(* IEC 61131-3 sources: elnaProjects/ElpcLogic/PomarKc7Changed/build_USO_ecl/_, 1 file *)

(* ---- plc.st ---- *)
TYPE
  TYPE_DualStateImAction : (_on, _off);
  TYPE_PhaseAlgoritmAction : (_run, _reset);
  TYPE_basketStats : STRUCT
    BASKET_NOTDEFINED : BYTE := 0;
    BASKET_ROLLEDIN : BYTE := 1;
    BASKET_ROLLEDOUT : BYTE := 2;
    BASKET_TRANSITIONAL : BYTE := 3;
    BASKET_ERROR : BYTE := 4;
    BASKET_TEST : BYTE := 5;
  END_STRUCT;
  TYPE_Answers : STRUCT
    ANS_NONE : UINT := 0;
    ANS_YES : UINT := 1;
    ANS_NO : UINT := 2;
    ANS_CANCEL : UINT := 4;
    ANS_RETRY : UINT := 8;
  END_STRUCT;
  struct_OilPump : STRUCT
    inCommand : WORD;
    inCommand_Alg : WORD;
    inCommand_ARM : WORD;
    status : DWORD;
    onStatus : BYTE;
    inOpcCommandsDisabled : BOOL;
    sdvig : BOOL;
    Ns : BOOL;
    CommandFault : BOOL;
    Accident : BOOL;
    Local : BOOL;
    Distance : BOOL;
    BreakCmdOn : BOOL;
    BreakCmdOff : BOOL;
    OpcCommandsDisabled : BOOL;
    lastCmdIsOn : BOOL;
    ISVALIDREF_statOn : BOOL;
    ISVALIDREF_statOff : BOOL;
    ISVALIDREF_cmdOn : BOOL;
    ISVALIDREF_cmdOff : BOOL;
    ISVALIDREF_inBreakCmdOn : BOOL;
    ISVALIDREF_inBreakCmdOff : BOOL;
    inBlocked : BOOL;
    Blocked : BOOL;
    Osnovnoy : BOOL;
    Rezervny : BOOL;
    cmdOn : BOOL;
    cmdOff : BOOL;
    reliability : BOOL;
  END_STRUCT;
  struct_AlgTimers : STRUCT
    AutoPns_OffTimer : UINT;
    AutoPns_OnTimer : UINT;
    vibegPNS_Timer : UINT;
    NO_waitCloseKran : UINT;
    AO_waitKran : UINT;
    testPms_BreakTest : UINT;
    testdPmg_BreakTest : UINT;
    puskOilSystem_BreakPuskTimer_Poil : UINT;
    engineRun_BreakPuskTimer : UINT;
    filling_BreakPuskTimer : UINT;
    filling_waitAfterKran4 : UINT;
    filling_waitAfterKran5 : UINT;
    puskK_wait720 : UINT;
    puskV_wait600 : UINT;
    No_wait120 : UINT;
    No_wait600 : UINT;
    No_wait5 : UINT;
  END_STRUCT;
  struct_Question : STRUCT
    AnswerVariants : UINT;
    inCommand : WORD;
    ask : BOOL;
    reset : BOOL;
    status : DWORD;
    answer : UINT;
    OpcCommandsDisabled : BOOL;
    inOpcCommandsDisabled : BOOL;
  END_STRUCT;
  AlgoritmsQuestions : STRUCT
    vibegPNS_algContinue : struct_Question;
    testPms_algContinue : struct_Question;
    testdPmg_algContinue : struct_Question;
    puskK_questionFilling : struct_Question;
    puskK_questionUnload : struct_Question;
    puskV_questionEngine : struct_Question;
    puskV_questionMVoff : struct_Question;
    SemiAutoPusk_cmdRun1ph : struct_Question;
    SemiAutoPusk_cmdRun2ph : struct_Question;
    SemiAutoPusk_cmdRun3ph : struct_Question;
    SemiAutoPusk_cmdRun4ph : struct_Question;
  END_STRUCT;
  TYPE_commandDualInput : STRUCT
    CMD_ON : BYTE := 1;
    CMD_OFF : BYTE := 2;
    CMD_RESET : BYTE := 3;
  END_STRUCT;
  TYPE_CommandAnalog : STRUCT
    cmd_SetUstavki : WORD := 1;
    cmd_SetRemont : WORD := 2;
    cmd_ResetRemont : WORD := 3;
    cmd_kvitNotReliable : WORD := 4;
  END_STRUCT;
  struct_AnalogParametr : STRUCT
    inCommand : WORD;
    inCommand_Alg : WORD;
    inCommand_ARM : WORD;
    status : DWORD;
    newValue : LREAL;
    currentValue : LREAL;
    minVal : LREAL;
    maxVal : LREAL;
    maxStep : LREAL;
    minVal_ISVALIDREF : BOOL;
    maxVal_ISVALIDREF : BOOL;
    maxStep_ISVALIDREF : BOOL;
    inOpcCommandsDisabled : BOOL;
    Value : LREAL;
    isValidValue : BOOL;
    OpcCommandsDisabled : BOOL;
  END_STRUCT;
  struct_AI : STRUCT
    value : LREAL;
    status : DWORD;
    interval : BYTE;
    inCommand : WORD;
    blConnect : BOOL;
    dLL : LREAL;
    dHL : LREAL;
    dLA : LREAL;
    dHA : LREAL;
    dLW : LREAL;
    dHW : LREAL;
    LL : LREAL;
    HL : LREAL;
    LA : LREAL;
    HA : LREAL;
    LW : LREAL;
    HW : LREAL;
    ISVALIDREF_LA : BOOL;
    ISVALIDREF_HA : BOOL;
    ISVALIDREF_LW : BOOL;
    ISVALIDREF_HW : BOOL;
    inpLL : LREAL;
    inpHL : LREAL;
    CurrentShotCircuit : LREAL;
    CurrentBreakCircuit : LREAL;
    maxChangeSpeed : LREAL;
    maxChangeSpeedDown : LREAL;
    ChangeSpeed : LREAL;
    histeresis : LREAL;
    aperturFilter : LREAL;
    exponentialFilter : LREAL;
    rassoglasovanie : LREAL;
    OpcCommandsDisabled : BOOL;
    Disabled_LA : BOOL;
    Disabled_HA : BOOL;
    Disabled_LW : BOOL;
    Disabled_HW : BOOL;
    delayLA : TIME;
    delayLW : TIME;
    delayHW : TIME;
    delayHA : TIME;
    minValue_ISVALIDREF : BOOL;
    maxValue_ISVALIDREF : BOOL;
    minValue : LREAL;
    maxValue : LREAL;
    inOpcCommandsDisabled : BOOL;
    imit : BOOL;
    remont : BOOL;
    NS : BOOL;
    NS_Min : BOOL;
    NS_Max : BOOL;
    inCommand_Alg : WORD;
    inCommand_ARM : WORD;
    dMaxChangeSpeed : LREAL;
    dMaxChangeSpeedDown : LREAL;
  END_STRUCT;
  AiConfig : STRUCT
    Tstali_statora_kanal_1 : struct_AI;
    Tstali_statora_kanal_2 : struct_AI;
    Tstali_statora_kanal_3 : struct_AI;
    Tmedi_statora_kanal_1 : struct_AI;
    Tmedi_statora_kanal_2 : struct_AI;
    Tmedi_statora_kanal_3 : struct_AI;
    Toporno_podshipnika_EDT_1 : struct_AI;
    Toy_podshipnika_EDT_2 : struct_AI;
    Toy_podshipnika_kol_EDT_3 : struct_AI;
    Toy_podshipnika_kol_EDT_4 : struct_AI;
    Toy_podshipnika_shest_red_EDT_5 : struct_AI;
    Ty_podshipnika_red_EDT_6 : struct_AI;
    Ty_podshipnika_nagnet_EDT_7_1 : struct_AI;
    Ty_podshipnika_nagnet_EDT_7_2 : struct_AI;
    Toy_podshipnika_svobod_konca_EDT_8_1 : struct_AI;
    Toy_podshipnika_svobod_konca_EDT_8_2 : struct_AI;
    Toy_podshipnika_rab_kol_EDT_9_1 : struct_AI;
    Toy_podshipnika_rab_kol_EDT_9_2 : struct_AI;
    Toy_podshipnika_nerab_kol_EDT_10_1 : struct_AI;
    Toy_podshipnika_nerab_kol_EDT_10_2 : struct_AI;
    Tholodnogo_vozduha_ED_kanal_1 : struct_AI;
    Tholodnogo_vozduha_ED_kanal_2 : struct_AI;
    Tgorjachego_vozduha_ED_kanal_1 : struct_AI;
    Tgorjachego_vozduha_ED_kanal_2 : struct_AI;
    Tnarujnogo_vozduha : struct_AI;
    Tgaza_na_vhode_H : struct_AI;
    Tgaza_na_vyhode_H : struct_AI;
    Tmasla_do_AVOM : struct_AI;
    Tmasla_posle_AVOM : struct_AI;
    Tmasla_MB : struct_AI;
    Tmasla_MB_TEN : struct_AI;
    Tshu : struct_AI;
    Pmaslo_sm_nizkoe : struct_AI;
    Pmaslo_sm_vysokoe : struct_AI;
    Pmasla_posle_GNS : struct_AI;
    Pmasla_posle_NU : struct_AI;
    Pgaza_na_vhode_nagnetatelia : struct_AI;
    Pgaza_na_vyhode_nagnetatelia : struct_AI;
    Pimpuls_gaz : struct_AI;
    dPgaza_na_maslo_filtre : struct_AI;
    dPgaza_na_konfuzore : struct_AI;
    dPmaslo_gaz : struct_AI;
    Os_sdvig_nagnetatelja_plus : struct_AI;
    Os_sdvig_nagnetatelja_minus : struct_AI;
    Yroven_masla_MB : struct_AI;
    Kontrol_per_220V : struct_AI;
    Kontrol_post_220V : struct_AI;
    Tok_statora : struct_AI;
    Vibro_skorost_OPED_T1 : struct_AI;
    Vibro_skorost_OYPED_T2 : struct_AI;
    Vibro_skorost_OYP_kolesa_ED_T3 : struct_AI;
    Vibro_skorost_OP_kolesa_RH_T4 : struct_AI;
    Vibro_skorost_OP_shesterni_RED_T5 : struct_AI;
    Vibro_skorost_OP_shesterni_RED_T6 : struct_AI;
  END_STRUCT;
  struct_singleOutput : STRUCT
    wait_time : TIME;
    inCommand : WORD;
    inOpcCommandsDisabled : BOOL;
    Q : BOOL;
    status : DWORD;
    OpcCommandsDisabled : BOOL;
    inCommand_Alg : WORD;
    inCommand_ARM : WORD;
  END_STRUCT;
  IM_singleOutputs : STRUCT
    Rabota_EGPA : struct_singleOutput;
    Neispr_EGPA : struct_singleOutput;
    Avary_EGPA : struct_singleOutput;
    U_lamp_SHU : struct_singleOutput;
    AO_knopka_ind : struct_singleOutput;
    Pusk_SHUP : struct_singleOutput;
    Stop_SHUP : struct_singleOutput;
    NO_fonar : struct_singleOutput;
    PC_fonar : struct_singleOutput;
    AC_fonar : struct_singleOutput;
    Kr1_smazka : struct_singleOutput;
    Kr2_smazka : struct_singleOutput;
    Kr4_open_from_alg : struct_singleOutput;
    Synch_rej_K1 : struct_singleOutput;
  END_STRUCT;
  struct_Alg : STRUCT
    inRunOnStart : BOOL;
    inCanRun : BOOL;
    inHasError : BOOL;
    inEnded : BOOL;
    inOpcCommandsDisabled : BOOL;
    inCommand : WORD;
    inCommand_ARM : WORD;
    inCommand_Alg : WORD;
    status : DWORD;
    CanRun : BOOL;
    OpcCommandsDisabled : BOOL;
    isRuning : BOOL;
    HasError : BOOL;
    isEnded : BOOL;
    RunOnStart : BOOL;
    Start : DWORD;
    Error : DWORD;
    Top : DWORD;
  END_STRUCT;
  AlgoritmsConfig : STRUCT
    autoNu : struct_Alg;
    AutoPns : struct_Alg;
    AutoAvom : struct_Alg;
    AutoTen : struct_Alg;
    AntiPompag : struct_Alg;
    testIm : struct_Alg;
    TestProtection : struct_Alg;
    Remont : struct_Alg;
    ppu : struct_Alg;
    puskOilSystem : struct_Alg;
    engineRun : struct_Alg;
    filling : struct_Alg;
    LineToRing : struct_Alg;
    RingToLine : struct_Alg;
    Apusk : struct_Alg;
    SemiAutoPusk : struct_Alg;
    no : struct_Alg;
    vibegPNS : struct_Alg;
    ao : struct_Alg;
    testPms : struct_Alg;
    testdPmg : struct_Alg;
    puskV : struct_Alg;
    puskK : struct_Alg;
    Pusk_F_faza1 : struct_Alg;
    Pusk_F_faza2 : struct_Alg;
    Pusk_TH_faza : struct_Alg;
    Prov_PMS_ALG : struct_Alg;
    Prov_opressovka_ALG : struct_Alg;
    Pusk_SEC_faza_chastotny : struct_Alg;
    Pusk_SEC_faza_reactor : struct_Alg;
  END_STRUCT;
  TItemDIN : STRUCT
    wFlags : UINT := 0;
    wValue : UINT := 0;
    nanosec : ULINT := 0;
    reserve : ULINT := 0;
  END_STRUCT;
  TItemAIN : STRUCT
    wFlags : UINT := 0;
    wReserved : UINT := 0;
    dblValue : LREAL := 0.0;
    nanosec : ULINT := 0;
    reserve : ULINT := 0;
  END_STRUCT;
  struct_ReserveIM : STRUCT
    var1 : BOOL;
    var2 : BOOL;
  END_STRUCT;
  TYPE_ReliableBit : STRUCT
    value : BOOL;
    reliability : BOOL;
    _inversed : BOOL;
  END_STRUCT;
  struct_DI : STRUCT
    imit : BOOL;
    value : WORD;
    reliability : WORD;
    bits : ARRAY [0..15] OF TYPE_ReliableBit;
    blConnect : BOOL;
  END_STRUCT;
  struct_Kran : STRUCT
    inCommand : WORD;
    status : DWORD;
    onStatus : BYTE;
    inOpcCommandsDisabled : BOOL;
    sdvig : BOOL;
    Ns : BOOL;
    Dp : BOOL;
    CommandFault : BOOL;
    Accident : BOOL;
    Auto : BOOL;
    Manual : BOOL;
    Local : BOOL;
    Distance : BOOL;
    ErrorPowerOff : BOOL;
    ErrorBlock : BOOL;
    So : BOOL;
    Sz : BOOL;
    OpcCommandsDisabled : BOOL;
    lastCmdIsOn : BOOL;
    ISVALIDREF_statOn : BOOL;
    ISVALIDREF_statOff : BOOL;
    ISVALIDREF_cmdOn : BOOL;
    ISVALIDREF_cmdOff : BOOL;
    ISVALIDREF_inSo : BOOL;
    ISVALIDREF_inSz : BOOL;
    ISVALIDREF_inDp : BOOL;
    continueHoldCommand : TIME;
    inCommand_Alg : WORD;
    inCommand_ARM : WORD;
    cmdOn : BOOL;
    cmdOff : BOOL;
    reliability : BOOL;
  END_STRUCT;
  struct_Switch : STRUCT
    inCommand : WORD;
    status : DWORD;
    onStatus : BYTE;
    inOpcCommandsDisabled : BOOL;
    sdvig : BOOL;
    Ns : BOOL;
    CommandFault : BOOL;
    Accident : BOOL;
    Auto : BOOL;
    Manual : BOOL;
    Local : BOOL;
    Distance : BOOL;
    ErrorPowerOff : BOOL;
    ErrorBlock : BOOL;
    BreakCmdOn : BOOL;
    BreakCmdOff : BOOL;
    OpcCommandsDisabled : BOOL;
    lastCmdIsOn : BOOL;
    ISVALIDREF_statOn : BOOL;
    ISVALIDREF_statOff : BOOL;
    ISVALIDREF_cmdOn : BOOL;
    ISVALIDREF_cmdOff : BOOL;
    ISVALIDREF_inBreakCmdOn : BOOL;
    ISVALIDREF_inBreakCmdOff : BOOL;
    inCommand_Alg : WORD;
    inCommand_ARM : WORD;
    cmdOn : BOOL;
    cmdOff : BOOL;
    reliability : BOOL;
  END_STRUCT;
  struct_SectionSwitch : STRUCT
    inCommand : WORD;
    status : DWORD;
    onStatus : BYTE;
    inOpcCommandsDisabled : BOOL;
    sdvig : BOOL;
    Ns : BOOL;
    CommandFault : BOOL;
    Accident : BOOL;
    Local : BOOL;
    Distance : BOOL;
    OpcCommandsDisabled : BOOL;
    lastCmdIsOn : BOOL;
    offKNA : BOOL;
    basketStatus : BYTE;
    ISVALIDREF_statOn : BOOL;
    ISVALIDREF_statOff : BOOL;
    ISVALIDREF_cmdOn : BOOL;
    ISVALIDREF_cmdOff : BOOL;
    ISVALIDREF_inBreakCmdOn : BOOL;
    ISVALIDREF_inBreakCmdOff : BOOL;
    BreakCmdOn : BOOL;
    BreakCmdOff : BOOL;
    ISVALIDREF_basketRolledIn : BOOL;
    ISVALIDREF_basketRolledOut : BOOL;
    ISVALIDREF_basketTest : BOOL;
    inCommand_Alg : WORD;
    inCommand_ARM : WORD;
    cmdOn : BOOL;
    cmdOff : BOOL;
    reliability : BOOL;
  END_STRUCT;
  struct_ReserveIM2 : STRUCT
    var1 : BOOL;
    var2 : BOOL;
  END_STRUCT;
  struct_singleSignal : STRUCT
    reliability : BOOL;
    inverse : BOOL;
    DelayOn : TIME;
    DelayOff : TIME;
    Q : BOOL;
    status : DWORD;
    Disabled_Sig : BOOL;
  END_STRUCT;
  IM_singleSignals : STRUCT
    dP_maslo_gaz_Less100 : struct_singleSignal;
    dp_kran1_Less100 : struct_singleSignal;
    Razreshenie_zagruzki_dvig : struct_singleSignal;
    Vozbud_gotovnost : struct_singleSignal;
    Vozbud_neispr_tsepey_upr_AVR_pit : struct_singleSignal;
    Vozbud_neispravnost : struct_singleSignal;
    SHAVR1_v_rabote : struct_singleSignal;
    SHAVR2_v_rabote : struct_singleSignal;
    Avariinoe_otkluch_vikluchatelya : struct_singleSignal;
    Assinhronnii_hod_peregruzka : struct_singleSignal;
    SHU_v_GPA_vkluch : struct_singleSignal;
    SHP_v_GPA_vkluch : struct_singleSignal;
    QF1_on : struct_singleSignal;
    QF2_on : struct_singleSignal;
    QF23_on : struct_singleSignal;
    QF4_QF5_on : struct_singleSignal;
    QF6_QF7_on : struct_singleSignal;
    QF8_QF9_on : struct_singleSignal;
    QF10_QF11_on : struct_singleSignal;
    QF12_QF13_on : struct_singleSignal;
    QF14_QF15_on : struct_singleSignal;
    QF22_on : struct_singleSignal;
    NS_G1_G2 : struct_singleSignal;
    NS_G3_G4 : struct_singleSignal;
    NS_G15_G16 : struct_singleSignal;
    NS_G17 : struct_singleSignal;
    NS_G5_G6 : struct_singleSignal;
    NS_G7_G8 : struct_singleSignal;
    NS_G18_G19 : struct_singleSignal;
    NS_G10_G11 : struct_singleSignal;
    NS_G13_G14 : struct_singleSignal;
    Uroven_masla_akkum : struct_singleSignal;
    NKU1_GPA_on : struct_singleSignal;
    NKU2_GPA_on : struct_singleSignal;
    AO_KC_ot_SHKS : struct_singleSignal;
    AO_GPA_ot_SHU : struct_singleSignal;
    BEAO_srabotal : struct_singleSignal;
    Chastotny_pusk : struct_singleSignal;
    Neuspesh_chastotny_pusk : struct_singleSignal;
    Rezhim_ruchnogo_regulirovaniya : struct_singleSignal;
    Osnovnoy_regul_off : struct_singleSignal;
    Voltage_sekcii_norm : struct_singleSignal;
    Reactorny_pusk : struct_singleSignal;
    NO_GPA_ot_SHU : struct_singleSignal;
    AO_GPA_ot_PRU : struct_singleSignal;
    Nalichie_BP1 : struct_singleSignal;
    Nalichie_BP2 : struct_singleSignal;
    Nalichie_BP3 : struct_singleSignal;
    Nalichie_BP4 : struct_singleSignal;
    Nalichie_BP5 : struct_singleSignal;
    Nalichie_BP6 : struct_singleSignal;
    Nalichie_BP7_BP8 : struct_singleSignal;
    Nalichie_BP9_BP10 : struct_singleSignal;
    Nalichie_cepei_upravlen_mv : struct_singleSignal;
    Nalichie_220BEAO : struct_singleSignal;
    Nalichie_per_220_na_vhode : struct_singleSignal;
    Nalichie_post_220_na_vhode : struct_singleSignal;
    Nalichie_BP11 : struct_singleSignal;
    Nalichie_BP12 : struct_singleSignal;
    Dver_SHU_pered_otkrita : struct_singleSignal;
    Dver_SHU_zad_otkrita : struct_singleSignal;
    EO_GPA_ot_knopki_SHU : struct_singleSignal;
    EO_EGPA_ot_PRY : struct_singleSignal;
    Synchroniz_rezhima_K1 : struct_singleSignal;
    Potok_ms_posle_AVOM : struct_singleSignal;
  END_STRUCT;
  ImConfig : STRUCT
    Kran1 : struct_Kran;
    Kran2 : struct_Kran;
    Kran3 : struct_Kran;
    Kran3b : struct_Kran;
    Kran4 : struct_Kran;
    Kran5 : struct_Kran;
    Kran6 : struct_Kran;
    nu1 : struct_OilPump;
    nu2 : struct_OilPump;
    pns : struct_Switch;
    v1_Avom : struct_Switch;
    v2_Avom : struct_Switch;
    v3_Avom : struct_Switch;
    v4_Avom : struct_Switch;
    mv : struct_SectionSwitch;
    Reserve_IM1 : struct_ReserveIM;
    Reserve_IM2 : struct_ReserveIM2;
    SingleSignals : IM_singleSignals;
    SingleOutputs : IM_singleOutputs;
    KaloriferAVOM : struct_Switch;
    CMN : struct_Switch;
    TEN_kollectora : struct_Switch;
    TEN_MB : struct_Switch;
  END_STRUCT;
  TYPE_AnalogLimitFlags : STRUCT
    NONE : BYTE := 0;
    LL : BYTE := 16#1;
    LW : BYTE := 16#2;
    HW : BYTE := 16#4;
    LA : BYTE := 16#8;
    HA : BYTE := 16#10;
    HL : BYTE := 16#20;
    SipUP : BYTE := 16#40;
    SipDown : BYTE := 16#80;
  END_STRUCT;
  TWordData : STRUCT
    wFlags : UINT := 0;
    wValue : UINT := 0;
  END_STRUCT;
  struct_PhaseAlgoritm : STRUCT
    run : BOOL;
    reset : BOOL;
    start : BOOL;
    error : BOOL;
    top : BOOL;
    startStatus : DWORD;
    errorStatus : DWORD;
    topStatus : DWORD;
  END_STRUCT;
  struct_DO : STRUCT
    imit : BOOL;
    blConnect : BOOL;
    value : WORD;
    bits : ARRAY [0..15] OF BOOL;
  END_STRUCT;
  struct_AiProtection : STRUCT
    controlLimit : BYTE;
    delay : TIME;
    inTag : BYTE;
    inRunOnStart : BOOL;
    inCanRun : BOOL;
    inOpcCommandsDisabled : BOOL;
    inCommand : WORD;
    inCommand_Alg : WORD;
    inCommand_ARM : WORD;
    Tag : BYTE;
    status : DWORD;
    CanRun : BOOL;
    OpcCommandsDisabled : BOOL;
    isRunning : BOOL;
    HasError : BOOL;
    isEnded : BOOL;
    Remont : BOOL;
    Check : BOOL;
    Signaling : BOOL;
    SignalingTP : BOOL;
    RunOnStart : BOOL;
  END_STRUCT;
  TYPE_statusDualInput : STRUCT
    STATUS_NOTDEFINED : BYTE := 0;
    STATUS_ON : BYTE := 1;
    STATUS_OFF : BYTE := 2;
    STATUS_TRANSITIONAL : BYTE := 3;
    STATUS_ERROR : BYTE := 4;
  END_STRUCT;
  TYPE_StatusAi : STRUCT
    NOTDEFINED : BYTE := 0;
    LL : BYTE := 1;
    HL : BYTE := 2;
    NOTRELIABLE : BYTE := 3;
    normal : BYTE := 4;
    LW : BYTE := 5;
    HW : BYTE := 6;
    LA : BYTE := 7;
    HA : BYTE := 8;
  END_STRUCT;
  struct_DiProtection : STRUCT
    delay : TIME;
    inTag : BYTE;
    inRunOnStart : BOOL;
    inCanRun : BOOL;
    inOpcCommandsDisabled : BOOL;
    inCommand : WORD;
    inCommand_Alg : WORD;
    inCommand_ARM : WORD;
    Tag : BYTE;
    status : DWORD;
    CanRun : BOOL;
    OpcCommandsDisabled : BOOL;
    isRunning : BOOL;
    HasError : BOOL;
    isEnded : BOOL;
    Remont : BOOL;
    Check : BOOL;
    Signaling : BOOL;
    SignalingTP : BOOL;
    RunOnStart : BOOL;
  END_STRUCT;
  struct_AO : STRUCT
    nValue : LREAL;
    blConnect : BOOL;
    outLL : LREAL;
    outHL : LREAL;
    newLL : LREAL;
    newHL : LREAL;
    newLL_ISVALIDREF : BOOL;
    newHL_ISVALIDREF : BOOL;
    inCommand : WORD;
    Value : LREAL;
    status : DWORD;
    LL : LREAL;
    HL : LREAL;
    OpcCommandsDisabled : BOOL;
  END_STRUCT;
  AOConfig : STRUCT
    Reserv_AO_1 : struct_AO;
    Reserv_AO_2 : struct_AO;
  END_STRUCT;
  TYPE_ModeGpa : STRUCT
    MODE_NOTDEFINED : UINT := 0;
    MODE_REMONT : UINT := 1;
    MODE_STOP : UINT := 2;
    MODE_READY : UINT := 3;
    MODE_PUSKV : UINT := 4;
    MODE_PUSKK : UINT := 5;
    MODE_TESTDPMG : UINT := 6;
    MODE_TESTPMS : UINT := 7;
    MODE_APUSK : UINT := 8;
    MODE_MPUSK : UINT := 9;
    MODE_WORK_Ring : UINT := 10;
    MODE_WORK_Line : UINT := 11;
    MODE_NO : UINT := 12;
    MODE_AO : UINT := 13;
    MODE_EO : UINT := 14;
    MODE_TESTIM : UINT := 15;
    MODE_TESTAZ : UINT := 16;
    MODE_PUSK_FIRST_FAZA1 : UINT := 17;
    MODE_PUSK_FIRST_FAZA2 : UINT := 18;
  END_STRUCT;
  struct_DiscretParametr : STRUCT
    newValue : UINT;
    currentValue : UINT;
    inOpcCommandsDisabled : BOOL;
    inCommand : WORD;
    inCommand_Alg : WORD;
    inCommand_ARM : WORD;
    status : DWORD;
    OpcCommandsDisabled : BOOL;
    Value : UINT;
  END_STRUCT;
  struct_DualStateIm : STRUCT
    inCommand : WORD;
    status : DWORD;
    onStatus : BYTE;
    inOpcCommandsDisabled : BOOL;
    sdvig : BOOL;
    Ns : BOOL;
    CommandFault : BOOL;
    Accident : BOOL;
    OpcCommandsDisabled : BOOL;
    lastCmdIsOn : BOOL;
    ISVALIDREF_statOn : BOOL;
    ISVALIDREF_statOff : BOOL;
    ISVALIDREF_cmdOn : BOOL;
    ISVALIDREF_cmdOff : BOOL;
    inCommand_Alg : WORD;
    inCommand_ARM : WORD;
    cmdOn : BOOL;
    cmdOff : BOOL;
    reliability : BOOL;
  END_STRUCT;
  DiConfig : STRUCT
    di_0 : struct_DI;
    di_1 : struct_DI;
    di_2 : struct_DI;
    di_3 : struct_DI;
    di_4 : struct_DI;
    di_5 : struct_DI;
    di_6 : struct_DI;
    di_7 : struct_DI;
    di_8 : struct_DI;
    di_9 : struct_DI;
    di_10 : struct_DI;
    di_11 : struct_DI;
    di_12 : struct_DI;
    di_13 : struct_DI;
    di_14 : struct_DI;
    di_15 : struct_DI;
    di_16 : struct_DI;
    di_17 : struct_DI;
    di_18 : struct_DI;
    di_19 : struct_DI;
    di_20 : struct_DI;
    di_21 : struct_DI;
  END_STRUCT;
  TYPE_ProtectionTags : STRUCT
    NOTHING : BYTE := 0;
    AOB : BYTE := 1;
    AOS : BYTE := 2;
    AOPOJ : BYTE := 3;
  END_STRUCT;
  struct_AlgoritmsManager : STRUCT
    mode : UINT;
    narabotka : UINT;
    nMode : UINT;
    AnalogsPs : BOOL;
    DiscretPS : BOOL;
    ProtectionSignaling : BOOL;
  END_STRUCT;
  struct_ProtectionsManager : STRUCT
    inCommand : BYTE;
    protectionInRemont : BOOL;
  END_STRUCT;
  DOconfig : STRUCT
    do_0 : struct_DO;
    do_1 : struct_DO;
    do_2 : struct_DO;
    do_3 : struct_DO;
    do_4 : struct_DO;
    gpio_out : struct_DO;
  END_STRUCT;
  TYPE_TableRec : STRUCT
    x : REAL;
    y : REAL;
  END_STRUCT;
  TYPE_CommandsPotectionsManager : STRUCT
    RestartAllSignaling : BYTE := 1;
    RestartAllProtections : BYTE := 2;
    CheckProtections : BYTE := 3;
    ResetAllProtections : BYTE := 4;
  END_STRUCT;
  TDoubleData : STRUCT
    wFlags : UINT := 0;
    dblValue : LREAL := 0.0;
  END_STRUCT;
  ProtectionsConfig : STRUCT
    Topornogo_podshipnika_EDT_1 : struct_AiProtection;
    Toy_podshipnika_EDT_2 : struct_AiProtection;
    Toy_podshipnika_kol_EDT_3 : struct_AiProtection;
    Toy_podshipnika_kol_EDT_4 : struct_AiProtection;
    To_podshipnika_shest_red_EDT_5 : struct_AiProtection;
    To_podshipnika_shest_red_EDT_6 : struct_AiProtection;
    To_podshipnika_N_EDT_7 : struct_AiProtection;
    To_podshipnika_svob_konca_EDT_8 : struct_AiProtection;
    Ty_podshipnika_rab_kol_EDT_9 : struct_AiProtection;
    Typornogo_podshipnika_nerab_kolodok_HT_10 : struct_AiProtection;
    Tgaza_na_vyhode_H : struct_AiProtection;
    Os_sdvig_nagnetatelja_plus : struct_AiProtection;
    Os_sdvig_nagnetatelja_minus : struct_AiProtection;
    Pgaza_na_vyhode_nagnetatelia_GPA_STOP : struct_AiProtection;
    Pgaza_na_vhode_nagnetatelia_GPA_STOP : struct_AiProtection;
    Pgaza_na_vyhode_nagnetatelia : struct_AiProtection;
    dPmaslo_gaz : struct_AiProtection;
    Pmaslo_sm_nizkoe : struct_AiProtection;
    Pmaslo_sm_vysokoe : struct_AiProtection;
    Vibro_skorost_OPED_T1 : struct_AiProtection;
    Vibro_skorost_OPED_T2 : struct_AiProtection;
    Vibro_skorost_OYP_kolesa_ED_T3 : struct_AiProtection;
    Vibro_skorost_OP_kolesa_RH_T4 : struct_AiProtection;
    Vibro_skorost_OP_shesterni_RED_T5 : struct_AiProtection;
    Vibro_skorost_OP_shesterni_RED_T6 : struct_AiProtection;
    dPmaslo_gaz_less100 : struct_DiProtection;
    Reg_vozb_off : struct_DiProtection;
    Fail_chastotnii_pusk : struct_DiProtection;
    Off_avar_vikluchatel : struct_DiProtection;
    AOKC_SHKC : struct_DiProtection;
    AO_PRU : struct_DiProtection;
    AO_ot_SHU : struct_DiProtection;
    mvOff : struct_DiProtection;
    Kran1_sdvig : struct_DiProtection;
    Kran2_sdvig : struct_DiProtection;
  END_STRUCT;
END_TYPE

FUNCTION_BLOCK OPC_IM_GET
  VAR_EXTERNAL
    IM_Kran1_command : UDINT;
    IM_Kran2_command : UDINT;
    IM_Kran3_command : UDINT;
    IM_Kran3b_command : UDINT;
    IM_Kran4_command : UDINT;
    IM_Kran5_command : UDINT;
    IM_Kran6_command : UDINT;
    IM_nu1_command : UDINT;
    IM_nu2_command : UDINT;
    IM_pns_command : UDINT;
    IM_v1_Avom_command : UDINT;
    IM_v2_Avom_command : UDINT;
    IM_v3_Avom_command : UDINT;
    IM_v4_Avom_command : UDINT;
    IM_mv_command : UDINT;
    IM_Reserve_IM1_command : UDINT;
    IM_Reserve_IM2_command : UDINT;
    IM_SingleSignals_command : UDINT;
    IM_SingleOutputs_command : UDINT;
    IM_KaloriferAVOM_command : UDINT;
    IM_CMN_command : UDINT;
    IM_TEN_kollectora_command : UDINT;
    IM_TEN_MB_command : UDINT;
  END_VAR

  im.Kran1.inCommand_ARM := UINT_TO_WORD(IM_Kran1_command);

  im.Kran2.inCommand_ARM := UINT_TO_WORD(IM_Kran2_command);

  im.Kran3.inCommand_ARM := UINT_TO_WORD(IM_Kran3_command);

  im.Kran3b.inCommand_ARM := UINT_TO_WORD(IM_Kran3b_command);

  im.Kran4.inCommand_ARM := UINT_TO_WORD(IM_Kran4_command);

  im.Kran5.inCommand_ARM := UINT_TO_WORD(IM_Kran5_command);

  im.Kran6.inCommand_ARM := UINT_TO_WORD(IM_Kran6_command);

  im.nu1.inCommand_ARM := UINT_TO_WORD(IM_nu1_command);

  im.nu2.inCommand_ARM := UINT_TO_WORD(IM_nu2_command);

  im.pns.inCommand_ARM := UINT_TO_WORD(IM_pns_command);

  im.v1_Avom.inCommand_ARM := UINT_TO_WORD(IM_v1_Avom_command);

  im.v2_Avom.inCommand_ARM := UINT_TO_WORD(IM_v2_Avom_command);

  im.v3_Avom.inCommand_ARM := UINT_TO_WORD(IM_v3_Avom_command);

  im.v4_Avom.inCommand_ARM := UINT_TO_WORD(IM_v4_Avom_command);

  im.mv.inCommand_ARM := UINT_TO_WORD(IM_mv_command);

  im.KaloriferAVOM.inCommand_ARM := UINT_TO_WORD(IM_KaloriferAVOM_command);

  im.CMN.inCommand_ARM := UINT_TO_WORD(IM_CMN_command);

  im.TEN_kollectora.inCommand_ARM := UINT_TO_WORD(IM_TEN_kollectora_command);

  im.TEN_MB.inCommand_ARM := UINT_TO_WORD(IM_TEN_MB_command);
END_FUNCTION_BLOCK

FUNCTION_BLOCK OPC_algoritms_set
  VAR_EXTERNAL
    algoritms : AlgoritmsConfig;
    algManager_Mode : UINT;
    algoritms_AutoAvom_status : UDINT;
    algoritms_AutoPns_OffTimer : UINT;
    algoritms_AutoPns_OnTimer : UINT;
    algoritms_AutoPns_status : UDINT;
    algoritms_AutoTen_status : UDINT;
    algoritms_Remont_status : UDINT;
    algoritms_TestProtection_status : UDINT;
    algoritms_autoNu_NotHasRezervNU : BOOL;
    algoritms_autoNu_status : UDINT;
    algoritms_puskOilSystem_Error : UDINT;
    algoritms_puskOilSystem_Start : UDINT;
    algoritms_puskOilSystem_Top : UDINT;
    algoritms_puskOilSystem_status : UDINT;
    algoritms_testIm_status : UDINT;
    algoritms_vibegPNS_Error : UDINT;
    algoritms_vibegPNS_Start : UDINT;
    algoritms_vibegPNS_Top : UDINT;
    algoritms_vibegPNS_algContinue_status : UDINT;
    algoritms_vibegPNS_status : UDINT;
    algoritms_vibegPNS_waitVibeg_timer : UINT;
    protectManager_protectionInRemont : BOOL;
    algManager : struct_AlgoritmsManager;
    protectManager : struct_ProtectionsManager;
    NotHasRezervNU : BOOL;
    AlgTimers : struct_AlgTimers;
    AlgQuestions : AlgoritmsQuestions;
    algoritms_Apusk_Error : UDINT;
    algoritms_Apusk_Start : UDINT;
    algoritms_Apusk_Top : UDINT;
    algoritms_Apusk_status : UDINT;
    algoritms_RingToLine_Error : UDINT;
    algoritms_RingToLine_Start : UDINT;
    algoritms_RingToLine_Top : UDINT;
    algoritms_RingToLine_status : UDINT;
    algoritms_SemiAutoPusk_Error : UDINT;
    algoritms_SemiAutoPusk_Start : UDINT;
    algoritms_SemiAutoPusk_Top : UDINT;
    algoritms_SemiAutoPusk_cmdRun1ph_status : UDINT;
    algoritms_SemiAutoPusk_cmdRun2ph_status : UDINT;
    algoritms_SemiAutoPusk_cmdRun3ph_status : UDINT;
    algoritms_SemiAutoPusk_cmdRun4ph_status : UDINT;
    algoritms_SemiAutoPusk_status : UDINT;
    algoritms_ao_Error : UDINT;
    algoritms_ao_Start : UDINT;
    algoritms_ao_Top : UDINT;
    algoritms_ao_status : UDINT;
    algoritms_ao_waitKran_timer : UINT;
    algoritms_engineRun_BreakPuskTimer_timer : UINT;
    algoritms_engineRun_Error : UDINT;
    algoritms_engineRun_Start : UDINT;
    algoritms_engineRun_Top : UDINT;
    algoritms_engineRun_status : UDINT;
    algoritms_filling_BreakPuskTimer_timer : UINT;
    algoritms_filling_Error : UDINT;
    algoritms_filling_Start : UDINT;
    algoritms_filling_Top : UDINT;
    algoritms_filling_status : UDINT;
    algoritms_filling_waitAfterKran4_timer : UINT;
    algoritms_filling_waitAfterKran5_timer : UINT;
    algoritms_no_Error : UDINT;
    algoritms_no_Start : UDINT;
    algoritms_no_Top : UDINT;
    algoritms_no_status : UDINT;
    algoritms_no_waitCloseKran_timer : UINT;
    algoritms_ppu_Error : UDINT;
    algoritms_ppu_Start : UDINT;
    algoritms_ppu_Top : UDINT;
    algoritms_ppu_status : UDINT;
    algoritms_puskK_Error : UDINT;
    algoritms_puskK_Start : UDINT;
    algoritms_puskK_Top : UDINT;
    algoritms_puskK_questionFilling_status : UDINT;
    algoritms_puskK_questionUnload_status : UDINT;
    algoritms_puskK_status : UDINT;
    algoritms_puskK_wait720_timer : UINT;
    algoritms_puskOilSystem_BreakPuskTimer_Poil_timer : UINT;
    algoritms_puskOilSystem_BreakPuskTimer_dPmg_timer : UINT;
    algoritms_puskV_Error : UDINT;
    algoritms_puskV_Start : UDINT;
    algoritms_puskV_Top : UDINT;
    algoritms_puskV_questionFilling_status : UDINT;
    algoritms_puskV_questionMVoff_status : UDINT;
    algoritms_puskV_status : UDINT;
    algoritms_puskV_wait600_timer : UINT;
    algoritms_testPms_BreakTest_timer : UINT;
    algoritms_testPms_Error : UDINT;
    algoritms_testPms_Start : UDINT;
    algoritms_testPms_Top : UDINT;
    algoritms_testPms_algContinue_status : UDINT;
    algoritms_testPms_status : UDINT;
    algoritms_testdPmg_BreakTest_timer : UINT;
    algoritms_testdPmg_Error : UDINT;
    algoritms_testdPmg_Start : UDINT;
    algoritms_testdPmg_Top : UDINT;
    algoritms_testdPmg_algContinue_status : UDINT;
    algoritms_testdPmg_status : UDINT;
  END_VAR

  (* OPC Set - algoritms. Запись текущих состояний тэгов _______________________________________________________*)

  algManager_Mode := algManager.mode;

  protectManager_protectionInRemont:= protectManager.protectionInRemont;

  algoritms_autoNu_NotHasRezervNU:= NotHasRezervNU;

  algoritms_no_Start	:= DWORD_TO_UDINT(algoritms.no.Start);
  algoritms_no_Error	:= DWORD_TO_UDINT(algoritms.no.Error);
  algoritms_no_Top	:= DWORD_TO_UDINT(algoritms.no.Top);
  algoritms_no_status	:= DWORD_TO_UDINT(algoritms.no.status);
  algoritms_no_waitCloseKran_timer	:= AlgTimers.NO_waitCloseKran;

  algoritms_ao_Start	:= DWORD_TO_UDINT(algoritms.ao.Start);
  algoritms_ao_Error	:= DWORD_TO_UDINT(algoritms.ao.Error);
  algoritms_ao_Top	:= DWORD_TO_UDINT(algoritms.ao.Top);
  algoritms_ao_status	:= DWORD_TO_UDINT(algoritms.ao.status);
  algoritms_ao_waitKran_timer	:= AlgTimers.AO_waitKran;

  algoritms_vibegPNS_Start		:= DWORD_TO_UDINT(algoritms.vibegPNS.Start);
  algoritms_vibegPNS_Error		:= DWORD_TO_UDINT(algoritms.vibegPNS.Error);
  algoritms_vibegPNS_Top		:= DWORD_TO_UDINT(algoritms.vibegPNS.Top);
  algoritms_vibegPNS_status		:= DWORD_TO_UDINT(algoritms.vibegPNS.status);
  algoritms_vibegPNS_waitVibeg_timer	:= AlgTimers.vibegPNS_Timer;
  algoritms_vibegPNS_algContinue_status	:= DWORD_TO_UDINT(AlgQuestions.vibegPNS_algContinue.status);

  algoritms_testPms_Start		:= DWORD_TO_UDINT(algoritms.testPms.Start);
  algoritms_testPms_Error		:= DWORD_TO_UDINT(algoritms.testPms.Error);
  algoritms_testPms_Top		:= DWORD_TO_UDINT(algoritms.testPms.Top);
  algoritms_testPms_status		:= DWORD_TO_UDINT(algoritms.testPms.status);
  algoritms_testPms_algContinue_status	:= DWORD_TO_UDINT(AlgQuestions.testPms_algContinue.status);
  algoritms_testPms_BreakTest_timer	:= AlgTimers.testPms_BreakTest;

  algoritms_testdPmg_Start		:= DWORD_TO_UDINT(algoritms.testdPmg.Start);
  algoritms_testdPmg_Error		:= DWORD_TO_UDINT(algoritms.testdPmg.Error);
  algoritms_testdPmg_Top		:= DWORD_TO_UDINT(algoritms.testdPmg.Top);
  algoritms_testdPmg_status		:= DWORD_TO_UDINT(algoritms.testdPmg.status);
  algoritms_testdPmg_algContinue_status	:= DWORD_TO_UDINT(AlgQuestions.testdPmg_algContinue.status);
  algoritms_testdPmg_BreakTest_timer	:= AlgTimers.testdPmg_BreakTest;

  algoritms_testIm_status	:= DWORD_TO_UDINT(algoritms.testIm.status);

  algoritms_ppu_status	:= DWORD_TO_UDINT(algoritms.ppu.status);
  algoritms_ppu_Start	          := DWORD_TO_UDINT(algoritms.ppu.Start);
  algoritms_ppu_Error	          := DWORD_TO_UDINT(algoritms.ppu.Error);
  algoritms_ppu_Top	          := DWORD_TO_UDINT(algoritms.ppu.Top);

  algoritms_puskOilSystem_status			:= DWORD_TO_UDINT(algoritms.puskOilSystem.status);
  algoritms_puskOilSystem_Start				:= DWORD_TO_UDINT(algoritms.puskOilSystem.Start);
  algoritms_puskOilSystem_Error				:= DWORD_TO_UDINT(algoritms.puskOilSystem.Error);
  algoritms_puskOilSystem_Top				:= DWORD_TO_UDINT(algoritms.puskOilSystem.Top);
  algoritms_puskOilSystem_BreakPuskTimer_Poil_timer	          := AlgTimers.puskOilSystem_BreakPuskTimer_Poil;

  algoritms_engineRun_status			:= DWORD_TO_UDINT(algoritms.engineRun.status);
  algoritms_engineRun_Start			:= DWORD_TO_UDINT(algoritms.engineRun.Start);
  algoritms_engineRun_Error			:= DWORD_TO_UDINT(algoritms.engineRun.Error);
  algoritms_engineRun_Top			:= DWORD_TO_UDINT(algoritms.engineRun.Top);
  algoritms_engineRun_BreakPuskTimer_timer	:= AlgTimers.engineRun_BreakPuskTimer;

  algoritms_filling_status		:= DWORD_TO_UDINT(algoritms.filling.status);
  algoritms_filling_Start		:= DWORD_TO_UDINT(algoritms.filling.Start);
  algoritms_filling_Error		:= DWORD_TO_UDINT(algoritms.filling.Error);
  algoritms_filling_Top		:= DWORD_TO_UDINT(algoritms.filling.Top);
  algoritms_filling_BreakPuskTimer_timer	:= AlgTimers.filling_BreakPuskTimer;
  algoritms_filling_waitAfterKran4_timer	:= AlgTimers.filling_waitAfterKran4;
  algoritms_filling_waitAfterKran5_timer	:= AlgTimers.filling_waitAfterKran5;

  algoritms_RingToLine_status	:= DWORD_TO_UDINT(algoritms.RingToLine.status);
  algoritms_RingToLine_Start	:= DWORD_TO_UDINT(algoritms.RingToLine.Start);
  algoritms_RingToLine_Error	:= DWORD_TO_UDINT(algoritms.RingToLine.Error);
  algoritms_RingToLine_Top	:= DWORD_TO_UDINT(algoritms.RingToLine.Top);

  algoritms_puskK_status	            := DWORD_TO_UDINT(algoritms.puskK.status);
  algoritms_puskK_Start	            := DWORD_TO_UDINT(algoritms.puskK.Start);
  algoritms_puskK_Error	            := DWORD_TO_UDINT(algoritms.puskK.Error);
  algoritms_puskK_Top	                      := DWORD_TO_UDINT(algoritms.puskK.Top);
  algoritms_puskK_wait720_timer	            := AlgTimers.puskK_wait720;
  algoritms_puskK_questionFilling_status	  := DWORD_TO_UDINT(AlgQuestions.puskK_questionFilling.status);
  algoritms_puskK_questionUnload_status	  := DWORD_TO_UDINT(AlgQuestions.puskK_questionUnload.status);

  algoritms_puskV_status	          := DWORD_TO_UDINT(algoritms.puskV.status);
  algoritms_puskV_Start	          := DWORD_TO_UDINT(algoritms.puskV.Start);
  algoritms_puskV_Error	          := DWORD_TO_UDINT(algoritms.puskV.Error);
  algoritms_puskV_Top	                    := DWORD_TO_UDINT(algoritms.puskV.Top);
  algoritms_puskV_wait600_timer	          := AlgTimers.puskV_wait600;
  algoritms_puskV_questionFilling_status	:= DWORD_TO_UDINT(AlgQuestions.puskV_questionEngine.status);
  algoritms_puskV_questionMVoff_status	:= DWORD_TO_UDINT(AlgQuestions.puskV_questionMVoff.status);

  algoritms_Apusk_status	:= DWORD_TO_UDINT(algoritms.Apusk.status);
  algoritms_Apusk_Start	:= DWORD_TO_UDINT(algoritms.Apusk.Start);
  algoritms_Apusk_Error	:= DWORD_TO_UDINT(algoritms.Apusk.Error);
  algoritms_Apusk_Top	          := DWORD_TO_UDINT(algoritms.Apusk.Top);

  algoritms_SemiAutoPusk_status	:= DWORD_TO_UDINT(algoritms.SemiAutoPusk.status);
  algoritms_SemiAutoPusk_Start	:= DWORD_TO_UDINT(algoritms.SemiAutoPusk.Start);
  algoritms_SemiAutoPusk_Error	:= DWORD_TO_UDINT(algoritms.SemiAutoPusk.Error);
  algoritms_SemiAutoPusk_Top	:= DWORD_TO_UDINT(algoritms.SemiAutoPusk.Top);
  algoritms_SemiAutoPusk_cmdRun1ph_status	:= DWORD_TO_UDINT(AlgQuestions.SemiAutoPusk_cmdRun1ph.status);
  algoritms_SemiAutoPusk_cmdRun2ph_status	:= DWORD_TO_UDINT(AlgQuestions.SemiAutoPusk_cmdRun2ph.status);
  algoritms_SemiAutoPusk_cmdRun3ph_status	:= DWORD_TO_UDINT(AlgQuestions.SemiAutoPusk_cmdRun3ph.status);
  algoritms_SemiAutoPusk_cmdRun4ph_status	:= DWORD_TO_UDINT(AlgQuestions.SemiAutoPusk_cmdRun4ph.status);

  algoritms_AutoPns_status	:= DWORD_TO_UDINT(algoritms.AutoPns.status);
  algoritms_AutoPns_OnTimer	:= AlgTimers.AutoPns_OnTimer;
  algoritms_AutoPns_OffTimer	:= AlgTimers.AutoPns_OffTimer;

  algoritms_autoNu_status	:= DWORD_TO_UDINT(algoritms.autoNu.status);

  algoritms_AutoAvom_status	:= DWORD_TO_UDINT(algoritms.AutoAvom.status);

  algoritms_TestProtection_status	:= DWORD_TO_UDINT(algoritms.TestProtection.status);

  algoritms_Remont_status	:= DWORD_TO_UDINT(algoritms.Remont.status);

  algoritms_AutoTen_status	:= DWORD_TO_UDINT(algoritms.AutoTen.status);
END_FUNCTION_BLOCK

FUNCTION runIfNotRunning : BOOL
  VAR_IN_OUT
    alg : struct_Alg;
  END_VAR
  VAR CONSTANT
    cmdRun : WORD      := 1;
  END_VAR

  IF NOT alg.isRuning THEN
                      alg.inOpcCommandsDisabled:=TRUE;
                      alg.inCanRun:=TRUE;
  		alg.inCommand_Alg:=cmdRun;
  END_IF;
END_FUNCTION

FUNCTION resetIfRunning : BOOL
  VAR_IN_OUT
    alg : struct_Alg;
  END_VAR
  VAR CONSTANT
    cmdReset : WORD      := 2;
  END_VAR

  IF alg.isRuning THEN
                      alg.inOpcCommandsDisabled:=TRUE;
  		alg.inCommand_Alg:=cmdReset;
  END_IF;
END_FUNCTION

FUNCTION_BLOCK fb_ph_algoritm
  VAR_IN_OUT
    alg : struct_Alg;
  END_VAR
  VAR_INPUT
    act : TYPE_PhaseAlgoritmAction;
    PhaseNumber : UINT;
    waitCompletion : BOOL;
  END_VAR
  VAR_IN_OUT
    StrPh : struct_PhaseAlgoritm;
  END_VAR
  VAR
    CommandFault_Trig : R_TRIG;
    reset_Trig : R_TRIG;
    _statusDualInput : TYPE_statusDualInput;
  END_VAR

  IF StrPh.run AND NOT StrPh.start THEN
  	StrPh.start := TRUE;
  	StrPh.top := FALSE;
  	StrPh.error := FALSE;
            StrPh.run:=FALSE;

  	CASE act OF
  		(*PhaseAlgoritmAction.run*)    _run : runIfNotRunning(alg); (*cmd_run*)
  		(*PhaseAlgoritmAction.reset*)_reset : resetIfRunning(alg); (*cmd_reset*)
  	END_CASE;
  END_IF;

  IF StrPh.start AND NOT StrPh.top THEN
                      CommandFault_Trig(CLK := alg.hasError);
                      IF CommandFault_Trig.Q THEN
  	          StrPh.error := TRUE;
                      END_IF;

  		CASE act OF
  		(*PhaseAlgoritmAction.run*)    _run:
                                                          IF waitCompletion THEN
  		                                	StrPh.top:=alg.isEnded;
  		                                    ELSE
  			                              StrPh.top:=alg.isRuning;
  		                                    END_IF;

  		(*PhaseAlgoritmAction.reset*) _reset:   StrPh.top := NOT alg.isRuning;
  		END_CASE;

  END_IF;

  IF StrPh.top THEN
  StrPh.error := FALSE;
  END_IF;

  reset_Trig(CLK := StrPh.reset);
  IF reset_Trig.Q THEN
            IF waitCompletion THEN
            resetIfRunning(alg);
            END_IF;
  	StrPh.start := FALSE;
  	StrPh.error := FALSE;
  	StrPh.top := FALSE;
            StrPh.run:=FALSE;
            StrPh.reset:=FALSE;
  END_IF;

  StrPh.startStatus := SHL(BOOL_TO_DWORD(StrPh.start), PhaseNumber);
  StrPh.errorStatus := SHL(BOOL_TO_DWORD(StrPh.error), PhaseNumber);
  StrPh.topStatus := SHL(BOOL_TO_DWORD(StrPh.top), PhaseNumber);
END_FUNCTION_BLOCK

FUNCTION_BLOCK fb_ph_Kran
  VAR_IN_OUT
    im : struct_Kran;
    StrPh : struct_PhaseAlgoritm;
  END_VAR
  VAR_INPUT
    act : TYPE_DualStateImAction;
    PhaseNumber : UINT;
  END_VAR
  VAR
    CommandFault_Trig : R_TRIG;
    reset_Trig : R_TRIG;
    _statusDualInput : TYPE_statusDualInput;
  END_VAR

  IF StrPh.run AND NOT StrPh.start THEN
  	StrPh.start := TRUE;
  	StrPh.top := FALSE;
  	StrPh.error := FALSE;
            StrPh.run:=FALSE;

  	CASE act OF
  		(*DualStateImAction.on*)   _on: im.inOpcCommandsDisabled:=TRUE;
                                                      im.inCommand_Alg := 1; (*cmd_open*)
  		(*DualStateImAction.off*) _off: im.inOpcCommandsDisabled:=TRUE;
                                                      im.inCommand_Alg := 2; (*cmd_close*)
  	END_CASE;
  END_IF;

  IF StrPh.start AND NOT StrPh.top THEN
                      CommandFault_Trig(CLK := im.CommandFault);
                      IF CommandFault_Trig.Q THEN
  	          StrPh.error := TRUE;
                      END_IF;

  		CASE act OF
  		(*_DualStateImAction.on*)    _on: StrPh.top := im.onStatus = _statusDualInput.STATUS_ON;
  		(*_DualStateImAction.off*)  _off: StrPh.top := im.onStatus = _statusDualInput.STATUS_OFF;
  		END_CASE;

  END_IF;

  IF StrPh.top THEN
  StrPh.error := FALSE;
  END_IF;

  reset_Trig(CLK := StrPh.reset);
  IF reset_Trig.Q THEN
  	StrPh.start := FALSE;
  	StrPh.error := FALSE;
  	StrPh.top := FALSE;
            StrPh.run:=FALSE;
            StrPh.reset:=FALSE;
  END_IF;

  StrPh.startStatus := SHL(BOOL_TO_DWORD(StrPh.start), PhaseNumber);
  StrPh.errorStatus := SHL(BOOL_TO_DWORD(StrPh.error), PhaseNumber);
  StrPh.topStatus := SHL(BOOL_TO_DWORD(StrPh.top), PhaseNumber);
END_FUNCTION_BLOCK

FUNCTION_BLOCK fb_ph_Timer
  VAR_INPUT
    delay : TIME;
    PhaseNumber : UINT;
  END_VAR
  VAR_IN_OUT
    StrPh : struct_PhaseAlgoritm;
  END_VAR
  VAR
    CommandFault_Trig : R_TRIG;
    reset_Trig : R_TRIG;
  END_VAR
  VAR_IN_OUT
    timer : UINT;
  END_VAR
  VAR
    _timer : TON;
    _statusDualInput : TYPE_statusDualInput;
  END_VAR

  IF StrPh.run AND NOT StrPh.start THEN
  	StrPh.start := TRUE;
  	StrPh.top := FALSE;
  	StrPh.error := FALSE;
            StrPh.run:=FALSE;

  END_IF;

  _timer(IN:=StrPh.start, PT:=delay);

  timer:=TIME_TO_UINT(delay -_timer.ET);

  IF StrPh.start AND NOT StrPh.top THEN
  StrPh.top:=_timer.Q;
  END_IF;

  reset_Trig(CLK := StrPh.reset);
  IF reset_Trig.Q THEN
  	StrPh.start := FALSE;
  	StrPh.error := FALSE;
  	StrPh.top := FALSE;
            StrPh.run:=FALSE;
            (*timer:=TIME_TO_UINT(delay -_timer.ET);*)
            StrPh.reset:=FALSE;
  END_IF;

  StrPh.startStatus := SHL(BOOL_TO_DWORD(StrPh.start), PhaseNumber);
  StrPh.errorStatus := SHL(BOOL_TO_DWORD(StrPh.error), PhaseNumber);
  StrPh.topStatus := SHL(BOOL_TO_DWORD(StrPh.top), PhaseNumber);
END_FUNCTION_BLOCK

FUNCTION_BLOCK fb_sunpackerCommand
  VAR_INPUT
    command : WORD;
  END_VAR
  VAR_OUTPUT
    source : BYTE;
    parametr : BYTE;
    cmd : BYTE;
  END_VAR

  cmd := WORD_TO_BYTE(command and 16#7);
  parametr := WORD_TO_BYTE(SHR((command and 16#1FF8), 3));
  source := WORD_TO_BYTE(SHR(command, 13));
END_FUNCTION_BLOCK

FUNCTION_BLOCK fb_Question
  VAR_IN_OUT
    StrQ : struct_Question;
  END_VAR
  VAR
    Asked : UINT;
    _answers : TYPE_Answers;
    _sunpackerCommand : fb_sunpackerCommand;
    source : BYTE;
    parametr : BYTE;
    lastParametr : BYTE;
    cmd : BYTE;
    source_for_Status : BYTE;
    cmd_for_Status : BYTE;
    command_error_for_Status : BYTE;
    resetCmdTimer : TON;
    resetCmdTimerPriznak : BOOL;
    reset_Trig : R_TRIG;
  END_VAR
  VAR CONSTANT
    cmd_answer : UINT      := 1;
  END_VAR

  StrQ.OpcCommandsDisabled := StrQ.inopcCommandsDisabled;

  IF StrQ.ask THEN
  StrQ.inopcCommandsDisabled:=FALSE;
      IF Asked=0 THEN
  	Asked:=StrQ.AnswerVariants;
  	StrQ.answer:=_answers.ANS_NONE;
      END_IF;

      _sunpackerCommand(command := StrQ.inCommand);
  	source := _sunpackerCommand.source;
            parametr := _sunpackerCommand.parametr;
  	cmd := _sunpackerCommand.cmd;

      IF cmd <> 0 AND lastParametr <> parametr AND ((NOT StrQ.OpcCommandsDisabled) AND source > 0)  then
  	CASE BYTE_TO_INT(cmd) OF
  	                               1 :

  				IF Asked<>0 THEN
                                             (* CASE BYTE_TO_INT(parametr) OF
                                              1: answer:=_answers.ANS_YES;
                                              2: answer:=_answers.ANS_NO;
                                              4: answer:=_answers.ANS_CANCEL;
                                              8: answer:=_answers.ANS_RETRY;
  	                                  END_CASE;*)
                                          StrQ.answer:=BYTE_TO_UINT(parametr);
                                          command_error_for_Status := 0;
                                          ELSE
  	                              command_error_for_Status := cmd;
                                          END_IF;
  	END_CASE;
  	source_for_Status := source;
  	cmd_for_Status := cmd;
  	resetCmdTimer(IN := FALSE);
  	resetCmdTimerPriznak := TRUE;
      END_IF;

      lastParametr := parametr;

      resetCmdTimer(IN := resetCmdTimerPriznak, PT := T#5S);
      IF resetCmdTimer.Q THEN
  	resetCmdTimerPriznak := FALSE;
  	source_for_Status := 0;
  	cmd_for_Status := 0;
  	command_error_for_Status := 0;
      END_IF;
  END_IF;

  reset_Trig(CLK := StrQ.reset);
  IF reset_Trig.Q THEN
  	Asked:=0;
  	StrQ.answer:=0;
            StrQ.ask:=FALSE;
            StrQ.reset:=FALSE;
  	StrQ.inopcCommandsDisabled:=TRUE;
  END_IF;

  StrQ.status := SHL(BYTE_TO_DWORD(source_for_Status), 29)
  			OR SHL(BYTE_TO_DWORD(cmd_for_Status), 26)
  			OR SHL(BYTE_TO_DWORD(command_error_for_Status), 23)
  			OR SHL(BOOL_TO_DWORD(StrQ.OpcCommandsDisabled ), 21);
  IF StrQ.answer = 0 THEN
      StrQ.status := StrQ.status  OR SHL(UINT_TO_DWORD(asked), 6);
  ELSE
      StrQ.status := StrQ.status  OR SHL(UINT_TO_DWORD(StrQ.answer), 6);
  END_IF;
END_FUNCTION_BLOCK

FUNCTION_BLOCK fb_ph_OilPump
  VAR_IN_OUT
    im : struct_OilPump;
  END_VAR
  VAR_INPUT
    act : TYPE_DualStateImAction;
    PhaseNumber : UINT;
  END_VAR
  VAR_IN_OUT
    StrPh : struct_PhaseAlgoritm;
  END_VAR
  VAR
    CommandFault_Trig : R_TRIG;
    reset_Trig : R_TRIG;
    _statusDualInput : TYPE_statusDualInput;
  END_VAR

  IF StrPh.run AND NOT StrPh.start THEN
  	StrPh.start := TRUE;
  	StrPh.top := FALSE;
  	StrPh.error := FALSE;

  	CASE act OF
  		(*DualStateImAction.on*)   _on :im.inOpcCommandsDisabled:=TRUE;
                                                      im.inCommand_Alg := 1; (*cmd_open*)
  		(*DualStateImAction.off*) _off :im.inOpcCommandsDisabled:=TRUE;
                                                      im.inCommand_Alg := 2; (*cmd_close*)
  	END_CASE;
  END_IF;

  IF StrPh.start OR StrPh.reset THEN
      StrPh.run:=FALSE;
  END_IF;

  IF StrPh.start AND NOT StrPh.top THEN
                      CommandFault_Trig(CLK := im.CommandFault);
                      IF CommandFault_Trig.Q THEN
  	          StrPh.error := TRUE;
                      END_IF;

  		CASE act OF
  		(*_DualStateImAction.on*)    _on: StrPh.top := im.onStatus = _statusDualInput.STATUS_ON;
  		(*_DualStateImAction.off*)  _off: StrPh.top := im.onStatus = _statusDualInput.STATUS_OFF;
  		END_CASE;

  END_IF;

  reset_Trig(CLK := StrPh.reset);
  IF reset_Trig.Q THEN
  	StrPh.start := FALSE;
  	StrPh.error := FALSE;
  	StrPh.top := FALSE;
            StrPh.reset:=FALSE;
  END_IF;

  StrPh.startStatus := SHL(BOOL_TO_DWORD(StrPh.start), PhaseNumber);
  StrPh.errorStatus := SHL(BOOL_TO_DWORD(StrPh.error), PhaseNumber);
  StrPh.topStatus := SHL(BOOL_TO_DWORD(StrPh.top), PhaseNumber);
END_FUNCTION_BLOCK

FUNCTION runDiProtection : BOOL
  VAR_IN_OUT
    protection : struct_DiProtection;
  END_VAR
  VAR CONSTANT
    cmdRun : WORD      := 1;
  END_VAR

  IF NOT protection.isRunning THEN
                      protection.inOpcCommandsDisabled:=TRUE;
  		protection.inCommand_Alg:=cmdRun;
  END_IF;
END_FUNCTION

FUNCTION resetAiProtection : BOOL
  VAR_IN_OUT
    protection : struct_AiProtection;
  END_VAR
  VAR CONSTANT
    cmdReset : WORD      := 2;
  END_VAR

  IF protection.isRunning THEN
                      protection.inOpcCommandsDisabled:=TRUE;
  		protection.inCommand_Alg:=cmdReset;
  END_IF;
END_FUNCTION

FUNCTION runAiProtection : BOOL
  VAR_IN_OUT
    protection : struct_AiProtection;
  END_VAR
  VAR CONSTANT
    cmdRun : WORD      := 1;
  END_VAR

  IF NOT protection.isRunning THEN
                      protection.inOpcCommandsDisabled:=TRUE;
  		protection.inCommand_Alg:=cmdRun;
  END_IF;
END_FUNCTION

FUNCTION runPhase : BOOL
  VAR_IN_OUT
    ph : struct_PhaseAlgoritm;
  END_VAR

  IF NOT ph.start THEN
                      ph.run:=TRUE;
  END_IF;
END_FUNCTION

FUNCTION resetPhase : BOOL
  VAR_IN_OUT
    ph : struct_PhaseAlgoritm;
  END_VAR

  IF ph.start OR ph.top THEN
                      ph.reset:=TRUE;
  END_IF;
END_FUNCTION

FUNCTION resetDiProtection : BOOL
  VAR_IN_OUT
    protection : struct_DiProtection;
  END_VAR
  VAR CONSTANT
    cmdReset : WORD      := 2;
  END_VAR

  IF protection.isRunning THEN
                      protection.inOpcCommandsDisabled:=TRUE;
  		protection.inCommand_Alg:=cmdReset;
  END_IF;
END_FUNCTION

FUNCTION_BLOCK Pusk_first_faza2
  VAR_IN_OUT
    StrAlg : struct_Alg;
  END_VAR
  VAR
    nu1On : struct_PhaseAlgoritm;
    nu2On : struct_PhaseAlgoritm;
    timer240 : struct_PhaseAlgoritm;
    dPmg_more100 : struct_PhaseAlgoritm;
    Auto_NU1 : struct_PhaseAlgoritm;
    Error_Alg : struct_PhaseAlgoritm;
    fb_timer240 : fb_ph_Timer;
    fb_nu1On : fb_ph_OilPump;
    fb_nu2On : fb_ph_OilPump;
    fb_dPmg_more100 : fb_ph_algoritm;
    fb_Auto_NU1 : fb_ph_algoritm;
    fb_Error_Alg : fb_ph_algoritm;
    _sunpackerCommand : fb_sunpackerCommand;
    _statusDualInput : TYPE_statusDualInput;
    _Answers : TYPE_Answers;
    source : BYTE;
    cmd : BYTE;
    lastCmd : BYTE;
    source_for_Status : BYTE;
    cmd_for_Status : BYTE;
    command_error_for_Status : BYTE;
    resetCmdTimer : TON;
    resetCmdTimerPriznak : BOOL;
    onInit : BOOL;
    waitReset : TON;
  END_VAR
  VAR_EXTERNAL
    ModeGpa : TYPE_ModeGpa;
    algManager : struct_AlgoritmsManager;
    IM : ImConfig;
    protections : ProtectionsConfig;
    algoritms : AlgoritmsConfig;
    ai : AiConfig;
  END_VAR
  VAR
    statusAi : TYPE_StatusAi;
  END_VAR

  IF NOT onInit THEN
           fb_nu1On(phaseNumber:=1, act:=_on );
           fb_nu2On(phaseNumber:=2, act:=_on);
           fb_dPmg_more100(phaseNumber:=3);
           fb_Error_Alg(phaseNumber:=4);
           fb_Auto_NU1(phaseNumber:=5);
  onInit:=TRUE;
  END_IF;

  fb_timer240(StrPh:=timer240);
  fb_nu1On(StrPh:= nu1On,Im:=Im.nu1);
  fb_nu2On(StrPh:= nu2On,Im:=Im.nu2);
  fb_dPmg_more100(StrPh:=dPmg_more100);
  fb_Auto_NU1(StrPh:=Auto_NU1, alg:=algoritms.autoNu); (*komu ono nujno to blat *)
  fb_Error_Alg(StrPh:=Error_Alg);

  StrAlg.CanRun := StrAlg.inCanRun;
  StrAlg.OpcCommandsDisabled := StrAlg.inOpcCommandsDisabled;

  IF StrAlg.isRuning THEN

      StrAlg.hasError := nu1On.error AND nu2On.error AND Auto_NU1.error;

      (* защита не возведена - запускаем таймер *)
      IF NOT dPmg_more100.top THEN
  	runPhase(timer240);
      END_IF;

      (* носос 1 не включен - включаем насос*)
      IF NOT nu1On.start THEN
  	runPhase(nu1On);
      END_IF;

      (* носос 2 не включен - включаем насос*)
      IF NOT nu2On.start THEN
  	runPhase(nu2On);
      END_IF;

      (* один из насосов включен - включение защиты *)
      IF ((IM.nu1.onStatus = _statusDualInput.status_on OR IM.nu2.onStatus = _statusDualInput.status_on) AND  (nu1On.start OR nu2On.Start)) THEN
  	runPhase(dPmg_more100);
  	nu1On.top:=TRUE;
            nu2On.top:=TRUE;
      END_IF;

      (* фаза защиты активна - включение защиты *)
      IF dPmg_more100.start AND NOT dPmg_more100.top THEN
  	IF NOT IM.SingleSignals.dP_maslo_gaz_Less100.Q AND IM.SingleSignals.dP_maslo_gaz_Less100.status = 1 AND
  	ai.dPmaslo_gaz.interval >= statusAi.normal AND ai.dPmaslo_gaz.value > 150.0 THEN
                dPmg_more100.top:=TRUE;
  	END_IF;
      END_IF;

      (*таймер завершился до возведения защит - ошибка *)
      IF timer240.top THEN
  	Error_Alg.error := TRUE;
      ELSE
  	Error_Alg.error := FALSE;
      END_IF;

      IF dPmg_more100.top AND nu1On.top AND nu2On.top THEN
  	Auto_NU1.top:=TRUE;
  	runAiProtection(protections.dPmaslo_gaz);
            runDiProtection(protections.dPmaslo_gaz_less100);
  	resetAiProtection(protections.Pgaza_na_vhode_nagnetatelia_GPA_STOP);
  	resetAiProtection(protections.Pgaza_na_vyhode_nagnetatelia_GPA_STOP);
  	algoritms.autoNu.CanRun:=TRUE;
  	(*algoritms.autoNu.run ();ниче не ясно*)
  	resetPhase(timer240);
      END_IF;
  END_IF;

  StrAlg.CanRun := StrAlg.inCanRun;
  StrAlg.OpcCommandsDisabled := StrAlg.inOpcCommandsDisabled;

  (* ---- Если управление с ВУ заблокировано, то  передаем команду из алгоритма ---- *)
  IF StrAlg.inOpcCommandsDisabled THEN
  	StrAlg.inCommand := StrAlg.inCommand_Alg;
  ELSE (* иначе передаем команду с АРМа*)
  	StrAlg.inCommand := StrAlg.inCommand_ARM;
  END_IF;

  _sunpackerCommand(command := StrAlg.inCommand);
  	source := _sunpackerCommand.source;
  	cmd := _sunpackerCommand.cmd;

  IF cmd <> 0 AND lastCmd <> cmd AND (((NOT StrAlg.opcCommandsDisabled) AND source > 0) OR source = 0) then
  	CASE BYTE_TO_INT(cmd) OF
  		(*cmdRun*) 1: 	IF (StrAlg.CanRun) THEN
  					StrAlg.isRuning := TRUE;
  					StrAlg.isEnded := FALSE;
  					StrAlg.hasError := FALSE;
  					(*****************       OnRun       *****************)
                                                    algManager.nMode:=ModeGpa.MODE_PUSK_FIRST_FAZA2;

                                                    runPhase(timer240);
                                                    runPhase(nu1On);
                                                    runPhase(nu2On);
                                                    resetAiProtection(protections.dPmaslo_gaz);
                                                    resetDiProtection(protections.dPmaslo_gaz_less100);

  					cmd_for_Status := cmd;
  					source_for_Status := source;
  					command_error_for_Status := 0;
  				ELSE
  					StrAlg.isRuning := FALSE;
  					StrAlg.isEnded := FALSE;
  					StrAlg.hasError := FALSE;

  					cmd_for_Status := 0;
  					source_for_Status := source;
  					command_error_for_Status := cmd;
  				END_IF;
  		(*cmdReset*) 2: 	StrAlg.isRuning := FALSE;
  				StrAlg.isEnded := FALSE;
  				StrAlg.hasError 	:= FALSE;

                                           (*****************       OnReset       *****************)
                                          waitReset(IN:=FALSE);
                                          StrAlg.inCanRun:=FALSE;

                                          resetPhase(nu1On);
                                          resetPhase(nu2On);
                                          resetPhase(timer240);
                                          resetPhase(dPmg_more100);
                                          resetPhase(Auto_NU1);
                                          resetPhase(Error_Alg);

                                          StrAlg.inOpcCommandsDisabled:=FALSE;

  				cmd_for_Status := cmd;
  				source_for_Status := source;
  				command_error_for_Status := 0;
  	END_CASE;
  	resetCmdTimer(IN := false);
  	resetCmdTimerPriznak := TRUE;
  END_IF;
  lastCmd := cmd;

  resetCmdTimer(IN := resetCmdTimerPriznak, PT := T#5S);
  IF resetCmdTimer.Q THEN
  	resetCmdTimerPriznak := FALSE;
  	source_for_Status := 0;
  	cmd_for_Status := 0;
  	command_error_for_Status := 0;
  END_IF;

  StrAlg.Start:= timer240.startStatus
              OR nu1On.startStatus
              OR nu2On.startStatus
              OR dPmg_more100.startStatus
              OR Auto_NU1.startStatus
              OR Error_Alg.startStatus;

  StrAlg.Error := timer240.errorStatus
              OR nu1On.errorStatus
              OR nu2On.errorStatus
              OR dPmg_more100.errorStatus
              OR Auto_NU1.errorStatus
              OR Error_Alg.errorStatus;

  StrAlg.Top := timer240.topStatus
              OR nu1On.topStatus
              OR nu2On.topStatus
              OR dPmg_more100.topStatus
              OR Auto_NU1.topStatus
              OR Error_Alg.topStatus;

  (*TODO: TYPE PROGRAM CODE HERE*)
  StrAlg.status :=  SHL(BYTE_TO_DWORD(source_for_Status), 29)
  			OR SHL(BYTE_TO_DWORD(cmd_for_Status), 26)
  			OR SHL(BYTE_TO_DWORD(command_error_for_Status), 23)
  			OR SHL(BOOL_TO_DWORD(StrAlg.OpcCommandsDisabled ), 21)
  			OR SHL(BOOL_TO_DWORD(StrAlg.hasError),4)
  			OR SHL(BOOL_TO_DWORD(StrAlg.CanRun),2)
  			OR SHL(BOOL_TO_DWORD(StrAlg.isEnded),1)
  			OR BOOL_TO_DWORD(StrAlg.isRuning);
END_FUNCTION_BLOCK

FUNCTION askQuestion : BOOL
  VAR_IN_OUT
    StrQ : struct_Question;
  END_VAR

  IF NOT StrQ.ask THEN
                      StrQ.inOpcCommandsDisabled:=FALSE;
                      StrQ.ask:=TRUE;
  END_IF;
END_FUNCTION

FUNCTION resetQuestion : BOOL
  VAR_IN_OUT
    StrQ : struct_Question;
  END_VAR

  IF StrQ.ask THEN
                      StrQ.inOpcCommandsDisabled:=TRUE;
                      StrQ.reset:=TRUE;
  END_IF;
END_FUNCTION

FUNCTION setValue : BOOL
  VAR_IN_OUT
    StrDP : struct_DiscretParametr;
  END_VAR
  VAR_INPUT
    newValue : UINT;
  END_VAR
  VAR
    cmd_ChangeValue : WORD      := 1;
  END_VAR

  StrDP.newValue:=newValue;
  StrDP.inOpcCommandsDisabled:=TRUE;
  StrDP.inCommand_Alg:=cmd_ChangeValue;
END_FUNCTION

FUNCTION_BLOCK Prov_opressovka
  VAR_IN_OUT
    StrAlg : struct_Alg;
  END_VAR
  VAR
    OPC_Control : struct_PhaseAlgoritm;
    Pms_more_50 : struct_PhaseAlgoritm;
    Pms_more_300 : struct_PhaseAlgoritm;
    dPmg_more_100 : struct_PhaseAlgoritm;
    P_zad : struct_PhaseAlgoritm;
    kran5Open : struct_PhaseAlgoritm;
    kran4Open : struct_PhaseAlgoritm;
    kran5Close : struct_PhaseAlgoritm;
    kran4Close : struct_PhaseAlgoritm;
    timer10 : struct_PhaseAlgoritm;
    P_vh_vyh_more_zad : struct_PhaseAlgoritm;
    Zapoln_Norm : struct_PhaseAlgoritm;
    First_Step : struct_PhaseAlgoritm;
    MaxZapolnenie_izm : REAL;
    Opressovka_Start : struct_Question;
    PNS_NU_ON_Ask : struct_Question;
    Zapolnit_kontur : struct_Question;
    fb_OPC_Control : fb_ph_algoritm;
    fb_Pms_more_50 : fb_ph_algoritm;
    fb_Pms_more_300 : fb_ph_algoritm;
    fb_dPmg_more_100 : fb_ph_algoritm;
    fb_P_zad : fb_ph_algoritm;
    fb_kran5Open : fb_ph_Kran;
    fb_kran4Open : fb_ph_Kran;
    fb_kran5Close : fb_ph_Kran;
    fb_kran4Close : fb_ph_Kran;
    fb_timer10 : fb_ph_Timer;
    fb_P_vh_vyh_more_zad : fb_ph_algoritm;
    fb_Zapoln_Norm : fb_ph_algoritm;
    fb_First_Step : fb_ph_algoritm;
    fb_Opressovka_Start : fb_Question;
    fb_PNS_NU_ON_Ask : fb_Question;
    fb_Zapolnit_kontur : fb_Question;
    onInit : BOOL;
  END_VAR
  VAR_EXTERNAL
    Im : ImConfig;
    ai : AiConfig;
  END_VAR
  VAR
    _sunpackerCommand : fb_sunpackerCommand;
    source : BYTE;
    cmd : BYTE;
    _statusDualInput : TYPE_statusDualInput;
    lastCmd : BYTE;
    _Answers : TYPE_Answers;
  END_VAR
  VAR_EXTERNAL
    ModeGpa : TYPE_ModeGpa;
    algManager : struct_AlgoritmsManager;
  END_VAR
  VAR
    cmd_for_Status : BYTE;
    source_for_Status : BYTE;
    command_error_for_Status : BYTE;
    resetCmdTimer : TON;
    waitReset : TON;
    resetCmdTimerPriznak : BOOL;
    _statusAi : TYPE_StatusAi;
    protections : ProtectionsConfig;
  END_VAR

  IF NOT onInit THEN
      fb_OPC_Control(phaseNumber:=1);
      fb_Pms_more_50(phaseNumber:=2);
      fb_Pms_more_300(phaseNumber:=3);
      fb_dPmg_more_100(phaseNumber:=4);
      fb_P_zad(phaseNumber:=5);
      fb_kran5Open(phaseNumber:=6, act:=_on);
      fb_kran4Open(phaseNumber:=7, act:=_on);
      fb_kran5Close(phaseNumber:=8, act:=_off);
      fb_kran4Close(phaseNumber:=9, act:=_off);
      fb_timer10(phaseNumber:=10, delay:=T#10S);
      fb_P_vh_vyh_more_zad(phaseNumber:=11);
      fb_Zapoln_Norm(phaseNumber:=12);
      fb_First_Step(phaseNumber:=13);
      Opressovka_Start.AnswerVariants:=_Answers.ANS_YES + _Answers.ANS_NO;
      PNS_NU_ON_Ask.AnswerVariants:=_Answers.ANS_YES;
      Zapolnit_kontur.AnswerVariants:=_Answers.ANS_YES;
      onInit:=TRUE;
  END_IF;

  fb_OPC_Control(StrPh:=OPC_Control);
  fb_Pms_more_50(StrPh:=Pms_more_50);
  fb_Pms_more_300(StrPh:=Pms_more_300);
  fb_dPmg_more_100(StrPh:=dPmg_more_100);
  fb_P_zad(StrPh:=P_zad);
  fb_kran5Open(StrPh:=kran5Open, Im:=Im.Kran5);
  fb_kran4Open(StrPh:=kran4Open, Im:=Im.Kran4);
  fb_kran5Close(StrPh:=kran5Close, Im:=Im.Kran5);
  fb_kran4Close(StrPh:=kran4Close, Im:=Im.Kran4);
  fb_timer10(StrPh:=timer10);
  fb_P_vh_vyh_more_zad(StrPh:=P_vh_vyh_more_zad);
  fb_Zapoln_Norm(StrPh:=Zapoln_Norm);
  fb_First_Step(StrPh:=First_Step);
  fb_Opressovka_Start(StrQ:=Opressovka_Start);
  fb_PNS_NU_ON_Ask(StrQ:=PNS_NU_ON_Ask);
  fb_Zapolnit_kontur(StrQ:=Zapolnit_kontur);

  StrAlg.CanRun := StrAlg.inCanRun;
  StrAlg.OpcCommandsDisabled := StrAlg.inOpcCommandsDisabled;

  IF StrAlg.isRuning THEN
     (*IF	algManager.mode <> ModeGpa.MODE_O THEN
  	    askQuestion(Opressovka_Start);
      END_IF;*)

      IF	Opressovka_Start.answer=_Answers.ANS_YES THEN
  	    askQuestion(Opressovka_Start);
  	    Im.kran6.inOpcCommandsDisabled := FALSE;
  	    (*algManager.setMode(nMode:=ModeGpa.MODE_O);*)
  	    runPhase(OPC_Control);
  	    resetAiProtection(protections.Pgaza_na_vyhode_nagnetatelia_GPA_STOP);
  	    resetAiProtection(protections.Pgaza_na_vhode_nagnetatelia_GPA_STOP);
          ELSIF Opressovka_Start.answer=_Answers.ANS_no THEN
                resetQuestion(Opressovka_Start);
      END_IF;

      IF	OPC_Control.start AND NOT OPC_Control.top THEN
  	    askQuestion(PNS_NU_ON_Ask);
      END_IF;
      IF	(PNS_NU_ON_Ask.answer=_Answers.ANS_YES) AND NOT OPC_Control.top THEN
  	    OPC_Control.top:=TRUE;
  	    resetQuestion(PNS_NU_ON_Ask);
      END_IF;

      IF	OPC_Control.top AND NOT Pms_more_50.start  THEN
  	    Im.pns.inOpcCommandsDisabled := FALSE;
  	    Im.kran6.inOpcCommandsDisabled := FALSE;
  	    runPhase(Pms_more_50);
  	    runPhase(Pms_more_300);
      END_IF;
      IF	OPC_Control.top AND Im.pns.onStatus = _statusDualInput.STATUS_On AND NOT dPmg_more_100.start THEN
  	    Im.nu1.inOpcCommandsDisabled := FALSE;
  	    Im.nu2.inOpcCommandsDisabled := FALSE;
  	    runPhase(dPmg_more_100);
      END_IF;

      IF	Im.nu1.onStatus = _statusDualInput.STATUS_On OR Im.nu2.onStatus = _statusDualInput.STATUS_On AND dPmg_more_100.start AND NOT dPmg_more_100.top THEN
  	    IF ai.dPmaslo_gaz.interval	>=	_statusAi.NORMAL AND
  		    ai.dPmaslo_gaz.value > 150.0 AND Im.SingleSignals.dP_maslo_gaz_Less100.reliability = TRUE AND NOT Im.SingleSignals.dP_maslo_gaz_Less100.Q THEN
  		    dPmg_more_100.top:=TRUE;
  		    runAiProtection(protections.dPmaslo_gaz);
  		    runDiProtection(protections.dPmaslo_gaz_less100);
  	    END_IF;
      END_IF;

      IF	Im.pns.onStatus = _statusDualInput.STATUS_On AND Pms_more_50.start AND NOT Pms_more_50.top THEN
  	        IF	ai.Pmaslo_sm_nizkoe.interval	>=	_statusAi.NORMAL AND
  		        ai.Pmaslo_sm_nizkoe.value > 50.0 THEN
  		        Pms_more_50.top:=TRUE;
                  runAiProtection(protections.Pmaslo_sm_nizkoe);
  	    END_IF;
      END_IF;

      IF	Im.pns.onStatus = _statusDualInput.STATUS_On AND Pms_more_300.start AND NOT Pms_more_300.top THEN
  	    IF	ai.Pmaslo_sm_vysokoe.interval	>=	_statusAi.NORMAL AND
  		    ai.Pmaslo_sm_vysokoe.value > 300.0 THEN
  		    Pms_more_300.top:=TRUE;
  		    runAiProtection(protections.Pmaslo_sm_vysokoe);
  	    END_IF;
      END_IF;

      (*IF	dPmg_more_100.top AND Pms_more_50.top AND Pms_more_300.top THEN
  	    CASE	Auto.value OF
  	    0:	Im.kran3.inOpcCommandsDisabled := FALSE;
  		Im.kran4.inOpcCommandsDisabled := FALSE;
  		Im.kran5.inOpcCommandsDisabled := FALSE;
  		Im.kran3b.inOpcCommandsDisabled := FALSE;
  		resetPhase(Zapolnit_kontur);
  		IF	Im.PerepadDavlenieKran1_Less100.Q THEN
  			Im.kran1.inOpcCommandsDisabled := FALSE;
  			Im.kran2.inOpcCommandsDisabled := FALSE;
  		ELSE
  			Im.kran1.inOpcCommandsDisabled := TRUE;
  			Im.kran2.inOpcCommandsDisabled := TRUE;
  		END_IF
  		resetPhase(P_vh_vyh_more_zad);
  		resetPhase(kran5Open);
  		resetPhase(kran4Open);
  		resetPhase(timer10);
  		resetPhase(kran5Close);
  		resetPhase(P_zad);
  		resetPhase(First_Step);
  		resetPhase(kran4Close);
  		(*MaxZapolnenie_izm:=0;
  		MaxZapolnenie.setValue (0);
  	1:
  		Zapoln_Norm.top:= MaxZapolnenie.value - MaxZapolnenie_izm > 0.4 AND MaxZapolnenie.value >= 0.4 AND MaxZapolnenie.value <= 10 AND
  			ai.DGazaNaVhodeNagnetatelja.interval >= _statusAi.NORMAL AND MaxZapolnenie.value - ai.DGazaNaVhodeNagnetatelja.value > 0.4 AND
  			ai.DGazaNaVyhodeNagnetatelja.interval >= _statusAi.NORMAL AND MaxZapolnenie.value - ai.DGazaNaVyhodeNagnetatelja.value > 0.4 *)
  		IF	kran4Close.top AND Zapoln_Norm.top AND NOT P_zad.start THEN
  			resetPhase(P_vh_vyh_more_zad);
  			resetPhase(kran5Open);
  			resetPhase(kran4Open);
  			resetPhase(timer10);
  			resetPhase(kran5Close);
  			resetPhase(kran4Close);
  		END_IF;
  		IF	NOT kran4Close.top OR kran4Close.top AND Zapoln_Norm.top AND NOT P_zad.start THEN
  		 	runPhase(P_zad);
  		END_IF;
  		IF NOT P_zad.top AND P_zad.start AND Zapoln_Norm.top THEN
  			askQuestion(Zapolnit_kontur);
  			Im.kran3.inOpcCommandsDisabled := TRUE;
  			Im.kran4.inOpcCommandsDisabled := TRUE;
  			Im.kran5.inOpcCommandsDisabled := TRUE;
  			Im.kran3b.inOpcCommandsDisabled := TRUE;
  			Im.kran1.inOpcCommandsDisabled := TRUE;
  			Im.kran2.inOpcCommandsDisabled := TRUE;

  		ELSIF NOT Zapoln_Norm.top AND NOT P_zad.top THEN
  				resetQuestion(Zapolnit_kontur);
  		END_IF;

          IF	(Zapolnit_kontur.answer=_Answers.ANS_YES) AND P_zad.start THEN
  			(*MaxZapolnenie_izm:= MaxZapolnenie.value;*)
  			IF 	NOT First_Step.top THEN
  				runPhase(kran5Open);
  			ELSE
  				runPhase(kran4Open);
  			END_IF;
  			resetQuestion(Zapolnit_kontur);
  			P_zad.top:=TRUE;
  		END_IF;
                      (*

  		IF	P_zad.top AND NOT kran4Close.top THEN
  			MaxZapolnenie.newvalue:=MaxZapolnenie_izm;
  		ELSE
  			MaxZapolnenie.newvalue:= MaxZapolnenie.newvalue;
  		END_IF;*)

  		IF	kran5Open.top AND NOT First_Step.top THEN
  			runPhase(kran4Open);
  		END_IF;

          IF 	kran4Open.top AND NOT timer10.top AND NOT First_Step.top THEN
  			runPhase(timer10);
  		END_IF;

  		IF	timer10.top AND NOT First_Step.top THEN
  			runPhase(kran5Close);
  		END_IF;

  		IF	kran5Close.top OR First_Step.top AND kran4Open.top THEN
  			runPhase(P_vh_vyh_more_zad);
          END_IF;

  		IF	ai.Pgaza_na_vhode_nagnetatelia.interval >= _statusAi.NORMAL (*AND ai.Pgaza_na_vhode_nagnetatelia.value >= MaxZapolnenie.value*) AND
  			ai.Pgaza_na_vyhode_nagnetatelia.interval >= _statusAi.NORMAL (*AND ai.Pgaza_na_vyhode_nagnetatelia.value >= MaxZapolnenie.value*) AND  P_vh_vyh_more_zad.start AND NOT P_vh_vyh_more_zad.top THEN
  			runPhase(kran4Close);
  			P_vh_vyh_more_zad.top:=TRUE;
  		END_IF;

  		IF	kran4Close.top THEN
  			First_Step.top:=TRUE;
  			Im.kran3.inOpcCommandsDisabled := FALSE;
  			Im.kran4.inOpcCommandsDisabled := FALSE;
  			Im.kran5.inOpcCommandsDisabled := FALSE;
  			Im.kran3b.inOpcCommandsDisabled := FALSE;

              IF	Zapoln_Norm.top THEN
  				resetPhase(P_zad);
  			END_IF;

              IF	Im.SingleSignals.dp_kran1_Less100.Q THEN
  				Im.kran1.inOpcCommandsDisabled := FALSE;
  				Im.kran2.inOpcCommandsDisabled := FALSE;
  			ELSE
  				Im.kran1.inOpcCommandsDisabled := TRUE;
  				Im.kran2.inOpcCommandsDisabled := TRUE;
  			END_IF;
  		ELSE
  			Im.kran1.inOpcCommandsDisabled := TRUE;
  			Im.kran2.inOpcCommandsDisabled := TRUE;
  	    END_IF;
          END_IF;
          (*END_CASE;
  END_IF;*)

  _sunpackerCommand(command := StrAlg.inCommand);
  	source := _sunpackerCommand.source;
  	cmd := _sunpackerCommand.cmd;

  IF cmd <> 0 AND lastCmd <> cmd AND (((NOT StrAlg.opcCommandsDisabled) AND source > 0) OR source = 0) then
  	CASE BYTE_TO_INT(cmd) OF
  		(*cm dRun*) 1: 	IF (StrAlg.CanRun) THEN
  					StrAlg.isRuning := TRUE;
  					StrAlg.isEnded := FALSE;
  					StrAlg.hasError := FALSE;
  					(*****************       OnRun       *****************)
                                                    algManager.nMode:=ModeGpa.MODE_PUSK_FIRST_FAZA2;

                                                    (*runPhase(timer120);
                                                    runPhase(timer5);
                                                    runPhase(Shup);
                                                    resetAiProtection(protections.dPmaslo_gaz);
                                                    resetDiProtection(protections.dPmaslo_gaz_less100);*)

  					cmd_for_Status := cmd;
  					source_for_Status := source;
  					command_error_for_Status := 0;
  				ELSE
  					StrAlg.isRuning := FALSE;
  					StrAlg.isEnded := FALSE;
  					StrAlg.hasError := FALSE;

  					cmd_for_Status := 0;
  					source_for_Status := source;
  					command_error_for_Status := cmd;
  				END_IF;
  		(*cmdReset*) 2: 	StrAlg.isRuning := FALSE;
  				StrAlg.isEnded := FALSE;
  				StrAlg.hasError 	:= FALSE;

                                           (*****************       OnReset       *****************)
                                          waitReset(IN:=FALSE);
                                          StrAlg.inCanRun:=FALSE;

                                          (*resetPhase(timer5);
                                          resetPhase(Shup);
                                          resetPhase(timer120);
                                          resetPhase(Net_Chast);
                                          resetPhase(mvOn);
                                          resetPhase(pGNSmore04);
                                          resetPhase(gotov_K_zagruzke);
                                          resetPhase(dPmg_Top);
                                          resetPhase(AutoPNS_Start);*)

                                          StrAlg.inOpcCommandsDisabled:=FALSE;

  				cmd_for_Status := cmd;
  				source_for_Status := source;
  				command_error_for_Status := 0;
  	END_CASE;
  	resetCmdTimer(IN := false);
  	resetCmdTimerPriznak := TRUE;
  END_IF;
  lastCmd := cmd;

  resetCmdTimer(IN := resetCmdTimerPriznak, PT := T#5S);
  IF resetCmdTimer.Q THEN
  	resetCmdTimerPriznak := FALSE;
  	source_for_Status := 0;
  	cmd_for_Status := 0;
  	command_error_for_Status := 0;
  END_IF;

  StrAlg.Start:= OPC_Control.startStatus
              OR Pms_more_50.startStatus
              OR Pms_more_300.startStatus
              OR dPmg_more_100.startStatus
              OR P_zad.startStatus
              OR kran5Open.startStatus
              OR kran4Open.startStatus
              OR kran5Close.startStatus
              OR kran4Close.startStatus
              OR timer10.startStatus
              OR P_vh_vyh_more_zad.startStatus
              OR Zapoln_Norm.startStatus
              OR First_Step.startStatus;

  StrAlg.Top :=  OPC_Control.topStatus
              OR Pms_more_50.topStatus
              OR Pms_more_300.topStatus
              OR dPmg_more_100.topStatus
              OR P_zad.topStatus
              OR kran5Open.topStatus
              OR kran4Open.topStatus
              OR kran5Close.topStatus
              OR kran4Close.topStatus
              OR timer10.topStatus
              OR P_vh_vyh_more_zad.topStatus
              OR Zapoln_Norm.topStatus
              OR First_Step.topStatus;

  StrAlg.Error :=  OPC_Control.errorStatus
              OR Pms_more_50.errorStatus
              OR Pms_more_300.errorStatus
              OR dPmg_more_100.errorStatus
              OR P_zad.errorStatus
              OR kran5Open.errorStatus
              OR kran4Open.errorStatus
              OR kran5Close.errorStatus
              OR kran4Close.errorStatus
              OR timer10.errorStatus
              OR P_vh_vyh_more_zad.errorStatus
              OR Zapoln_Norm.errorStatus
              OR First_Step.errorStatus;

  (*TODO: TYPE PROGRAM CODE HERE*)
  StrAlg.status :=  SHL(BYTE_TO_DWORD(source_for_Status), 29)
  			OR SHL(BYTE_TO_DWORD(cmd_for_Status), 26)
  			OR SHL(BYTE_TO_DWORD(command_error_for_Status), 23)
  			OR SHL(BOOL_TO_DWORD(StrAlg.OpcCommandsDisabled ), 21)
  			OR SHL(BOOL_TO_DWORD(StrAlg.hasError),4)
  			OR SHL(BOOL_TO_DWORD(StrAlg.CanRun),2)
  			OR SHL(BOOL_TO_DWORD(StrAlg.isEnded),1)
  			OR BOOL_TO_DWORD(StrAlg.isRuning);
END_FUNCTION_BLOCK

FUNCTION_BLOCK fb_ph_Switch
  VAR_IN_OUT
    im : struct_Switch;
  END_VAR
  VAR_INPUT
    act : TYPE_DualStateImAction;
    PhaseNumber : UINT;
  END_VAR
  VAR_IN_OUT
    StrPh : struct_PhaseAlgoritm;
  END_VAR
  VAR
    CommandFault_Trig : R_TRIG;
    reset_Trig : R_TRIG;
    _statusDualInput : TYPE_statusDualInput;
  END_VAR

  IF StrPh.run AND NOT StrPh.start THEN
  	StrPh.start := TRUE;
  	StrPh.top := FALSE;
  	StrPh.error := FALSE;
            StrPh.run:=FALSE;

  	CASE act OF
  		(*DualStateImAction.on*)   _on :im.inOpcCommandsDisabled:=TRUE;
                                                      im.inCommand_Alg := 1; (*cmd_open*)
  		(*DualStateImAction.off*) _off :im.inOpcCommandsDisabled:=TRUE;
                                                      im.inCommand_Alg := 2; (*cmd_close*)
  	END_CASE;
  END_IF;

  IF StrPh.start AND NOT StrPh.top THEN
                      CommandFault_Trig(CLK := im.CommandFault);
                      IF CommandFault_Trig.Q THEN
  	          StrPh.error := TRUE;
                      END_IF;

  		CASE act OF
  		(*_DualStateImAction.on*)    _on: StrPh.top := im.onStatus = _statusDualInput.STATUS_ON;
  		(*_DualStateImAction.off*)  _off: StrPh.top := im.onStatus = _statusDualInput.STATUS_OFF;
  		END_CASE;

  END_IF;

  IF StrPh.top THEN
  StrPh.error := FALSE;
  END_IF;

  reset_Trig(CLK := StrPh.reset);
  IF reset_Trig.Q THEN
  	StrPh.start := FALSE;
  	StrPh.error := FALSE;
  	StrPh.top := FALSE;
            StrPh.run:=FALSE;
            StrPh.reset:=FALSE;
  END_IF;

  StrPh.startStatus := SHL(BOOL_TO_DWORD(StrPh.start), PhaseNumber);
  StrPh.errorStatus := SHL(BOOL_TO_DWORD(StrPh.error), PhaseNumber);
  StrPh.topStatus := SHL(BOOL_TO_DWORD(StrPh.top), PhaseNumber);
END_FUNCTION_BLOCK

FUNCTION_BLOCK Prov_PMS
  VAR_IN_OUT
    StrAlg : struct_Alg;
  END_VAR
  VAR
    pnsOff : struct_PhaseAlgoritm;
    timer120 : struct_PhaseAlgoritm;
    Pms_less_25 : struct_PhaseAlgoritm;
    Pms_less_250 : struct_PhaseAlgoritm;
    Error_Alg : struct_PhaseAlgoritm;
    fb_Pms_less_25 : fb_ph_algoritm;
    fb_Pms_less_250 : fb_ph_algoritm;
    fb_pnsOff : fb_ph_Switch;
    fb_timer120 : fb_ph_Timer;
    fb_Error_Alg : fb_ph_algoritm;
    onInit : BOOL;
  END_VAR
  VAR_EXTERNAL
    Im : ImConfig;
    ai : AiConfig;
  END_VAR
  VAR
    _sunpackerCommand : fb_sunpackerCommand;
    source : BYTE;
    cmd : BYTE;
    _statusDualInput : TYPE_statusDualInput;
    lastCmd : BYTE;
    _Answers : TYPE_Answers;
  END_VAR
  VAR_EXTERNAL
    ModeGpa : TYPE_ModeGpa;
    algManager : struct_AlgoritmsManager;
  END_VAR
  VAR
    cmd_for_Status : BYTE;
    source_for_Status : BYTE;
    command_error_for_Status : BYTE;
    resetCmdTimer : TON;
    waitReset : TON;
    resetCmdTimerPriznak : BOOL;
    _statusAi : TYPE_StatusAi;
  END_VAR

  IF NOT onInit THEN
      fb_pnsOff(phaseNumber:=1, act:=_off);
      fb_timer120(phaseNumber:=2, delay:=T#120S);
      fb_Pms_less_25(phaseNumber:=3);
      fb_Pms_less_250(phaseNumber:=4);
      fb_Error_Alg(phaseNumber:=5);
      onInit:=TRUE;
  END_IF;

  fb_pnsOff(StrPh:=pnsOff, Im:=Im.pns);
  fb_timer120(StrPh:=timer120);
  fb_Pms_less_25(StrPh:=Pms_less_25);
  fb_Pms_less_250(StrPh:=Pms_less_250);
  fb_Error_Alg(StrPh:=Error_Alg);

  StrAlg.CanRun := StrAlg.inCanRun;
  StrAlg.OpcCommandsDisabled := StrAlg.inOpcCommandsDisabled;

  IF StrAlg.isRuning THEN
     (*IF NOT pnsOff.start THEN
  	    PNS_OFF_Ask.ask ();
      END_IF;
      IF	(PNS_OFF_Ask.answer=Answers.ANS_YES) THEN
  	    runPhase(pnsOff);
          PNS_OFF_Ask.reset ();
  	    IF NOT (Pms_less_250.top AND Pms_less_25.top) THEN
  	    	runPhase(timer120);
  	    END_IF;
      END_IF;*)

      (*запуск проверок давления*)
      IF	pnsOff.top  THEN
          runPhase(Pms_less_25);
  	    runPhase(Pms_less_250);
      END_IF;

      (*проверка давления масла низкое*)
      IF	Pms_less_25.start AND NOT Pms_less_25.top THEN
  	    IF 	ai.Pmaslo_sm_nizkoe.interval>=_statusAi.NORMAL AND ai.Pmaslo_sm_nizkoe.value < 25.0 THEN
  	  	    Pms_less_25.top:=TRUE;
  	    END_IF;
      END_IF;

      IF	Pms_less_250.start AND NOT Pms_less_250.top THEN
  	    IF	ai.Pmaslo_sm_vysokoe.interval>=_statusAi.NORMAL AND ai.Pmaslo_sm_vysokoe.value < 250.0 THEN
  	  	    Pms_less_250.top:=TRUE;
  	    END_IF;
      END_IF;

      (*ошибка заврешия алгоритма по таймеру*)
      IF	timer120.top THEN
  	    Error_Alg.ERROR := TRUE;
      ELSE
  	    Error_Alg.ERROR := FALSE;
      END_IF;

      (*если проверка прошла - сброс таймера *)
      IF	Pms_less_250.top AND Pms_less_25.top  THEN
          resetPhase(timer120);
      END_IF;
  END_IF;

  _sunpackerCommand(command := StrAlg.inCommand);
  	source := _sunpackerCommand.source;
  	cmd := _sunpackerCommand.cmd;

  IF cmd <> 0 AND lastCmd <> cmd AND (((NOT StrAlg.opcCommandsDisabled) AND source > 0) OR source = 0) then
  	CASE BYTE_TO_INT(cmd) OF
  		(*cm dRun*) 1: 	IF (StrAlg.CanRun) THEN
  					StrAlg.isRuning := TRUE;
  					StrAlg.isEnded := FALSE;
  					StrAlg.hasError := FALSE;
  					(*****************       OnRun       *****************)
                                                    algManager.nMode:=ModeGpa.MODE_PUSK_FIRST_FAZA2;

                                                    (*runPhase(timer120);
                                                    runPhase(timer5);
                                                    runPhase(Shup);
                                                    resetAiProtection(protections.dPmaslo_gaz);
                                                    resetDiProtection(protections.dPmaslo_gaz_less100);*)

  					cmd_for_Status := cmd;
  					source_for_Status := source;
  					command_error_for_Status := 0;
  				ELSE
  					StrAlg.isRuning := FALSE;
  					StrAlg.isEnded := FALSE;
  					StrAlg.hasError := FALSE;

  					cmd_for_Status := 0;
  					source_for_Status := source;
  					command_error_for_Status := cmd;
  				END_IF;
  		(*cmdReset*) 2: 	StrAlg.isRuning := FALSE;
  				StrAlg.isEnded := FALSE;
  				StrAlg.hasError 	:= FALSE;

                                           (*****************       OnReset       *****************)
                                          waitReset(IN:=FALSE);
                                          StrAlg.inCanRun:=FALSE;

                                          (*resetPhase(timer5);
                                          resetPhase(Shup);
                                          resetPhase(timer120);
                                          resetPhase(Net_Chast);
                                          resetPhase(mvOn);
                                          resetPhase(pGNSmore04);
                                          resetPhase(gotov_K_zagruzke);
                                          resetPhase(dPmg_Top);
                                          resetPhase(AutoPNS_Start);*)

                                          StrAlg.inOpcCommandsDisabled:=FALSE;

  				cmd_for_Status := cmd;
  				source_for_Status := source;
  				command_error_for_Status := 0;
  	END_CASE;
  	resetCmdTimer(IN := false);
  	resetCmdTimerPriznak := TRUE;
  END_IF;
  lastCmd := cmd;

  resetCmdTimer(IN := resetCmdTimerPriznak, PT := T#5S);
  IF resetCmdTimer.Q THEN
  	resetCmdTimerPriznak := FALSE;
  	source_for_Status := 0;
  	cmd_for_Status := 0;
  	command_error_for_Status := 0;
  END_IF;

  StrAlg.Start:= pnsOff.startStatus
              OR timer120.startStatus
              OR Pms_less_25.startStatus
              OR Pms_less_250.startStatus;

  StrAlg.Top :=  pnsOff.topStatus
              OR timer120.topStatus
              OR Pms_less_25.topStatus
              OR Pms_less_250.topStatus;

  StrAlg.Error :=  pnsOff.errorStatus
              OR timer120.errorStatus
              OR Pms_less_25.errorStatus
              OR Pms_less_250.errorStatus;

  (*TODO: TYPE PROGRAM CODE HERE*)
  StrAlg.status :=  SHL(BYTE_TO_DWORD(source_for_Status), 29)
  			OR SHL(BYTE_TO_DWORD(cmd_for_Status), 26)
  			OR SHL(BYTE_TO_DWORD(command_error_for_Status), 23)
  			OR SHL(BOOL_TO_DWORD(StrAlg.OpcCommandsDisabled ), 21)
  			OR SHL(BOOL_TO_DWORD(StrAlg.hasError),4)
  			OR SHL(BOOL_TO_DWORD(StrAlg.CanRun),2)
  			OR SHL(BOOL_TO_DWORD(StrAlg.isEnded),1)
  			OR BOOL_TO_DWORD(StrAlg.isRuning);
END_FUNCTION_BLOCK

FUNCTION_BLOCK OPC_algoritms_get
  VAR_EXTERNAL
    AI_autoNu_command : UINT;
    AI_AutoPns_command : UINT;
    AI_AutoAvom_command : UINT;
    AI_AutoTen_command : UINT;
    AI_AntiPompag_command : UINT;
    AI_testIm_command : UINT;
    AI_TestProtection_command : UINT;
    AI_Remont_command : UINT;
    AI_ppu_command : UINT;
    AI_puskOilSystem_command : UINT;
    AI_engineRun_command : UINT;
    AI_filling_command : UINT;
    AI_LineToRing_command : UINT;
    AI_RingToLine_command : UINT;
    AI_Apusk_command : UINT;
    AI_SemiAutoPusk_command : UINT;
    AI_no_command : UINT;
    AI_vibegPNS_command : UINT;
    AI_ao_command : UINT;
    AI_testPms_command : UINT;
    AI_testdPmg_command : UINT;
    AI_puskV_command : UINT;
    AI_puskK_command : UINT;
    AI_Pusk_F_faza1_command : UINT;
    AI_Pusk_F_faza2_command : UINT;
    AI_Pusk_TH_faza_command : UINT;
    AI_Prov_PMS_ALG_command : UINT;
    AI_Prov_opressovka_ALG_command : UINT;
    AI_Pusk_SEC_faza_chastotny_command : UINT;
    AI_Pusk_SEC_faza_reactor_command : UINT;
    algoritms : AlgoritmsConfig;
  END_VAR

  algoritms.autoNu.inCommand_ARM := UINT_TO_WORD(AI_autoNu_command);

  algoritms.AutoPns.inCommand_ARM := UINT_TO_WORD(AI_AutoPns_command);

  algoritms.AutoAvom.inCommand_ARM := UINT_TO_WORD(AI_AutoAvom_command);

  algoritms.AutoTen.inCommand_ARM := UINT_TO_WORD(AI_AutoTen_command);

  algoritms.AntiPompag.inCommand_ARM := UINT_TO_WORD(AI_AntiPompag_command);

  algoritms.testIm.inCommand_ARM := UINT_TO_WORD(AI_testIm_command);

  algoritms.TestProtection.inCommand_ARM := UINT_TO_WORD(AI_TestProtection_command);

  algoritms.Remont.inCommand_ARM := UINT_TO_WORD(AI_Remont_command);

  algoritms.ppu.inCommand_ARM := UINT_TO_WORD(AI_ppu_command);

  algoritms.puskOilSystem.inCommand_ARM := UINT_TO_WORD(AI_puskOilSystem_command);

  algoritms.engineRun.inCommand_ARM := UINT_TO_WORD(AI_engineRun_command);

  algoritms.filling.inCommand_ARM := UINT_TO_WORD(AI_filling_command);

  algoritms.LineToRing.inCommand_ARM := UINT_TO_WORD(AI_LineToRing_command);

  algoritms.RingToLine.inCommand_ARM := UINT_TO_WORD(AI_RingToLine_command);

  algoritms.Apusk.inCommand_ARM := UINT_TO_WORD(AI_Apusk_command);

  algoritms.SemiAutoPusk.inCommand_ARM := UINT_TO_WORD(AI_SemiAutoPusk_command);

  algoritms.no.inCommand_ARM := UINT_TO_WORD(AI_no_command);

  algoritms.vibegPNS.inCommand_ARM := UINT_TO_WORD(AI_vibegPNS_command);

  algoritms.ao.inCommand_ARM := UINT_TO_WORD(AI_ao_command);

  algoritms.testPms.inCommand_ARM := UINT_TO_WORD(AI_testPms_command);

  algoritms.testdPmg.inCommand_ARM := UINT_TO_WORD(AI_testdPmg_command);

  algoritms.puskV.inCommand_ARM := UINT_TO_WORD(AI_puskV_command);

  algoritms.puskK.inCommand_ARM := UINT_TO_WORD(AI_puskK_command);

  algoritms.Pusk_F_faza1.inCommand_ARM := UINT_TO_WORD(AI_Pusk_F_faza1_command);

  algoritms.Pusk_F_faza2.inCommand_ARM := UINT_TO_WORD(AI_Pusk_F_faza2_command);

  algoritms.Pusk_TH_faza.inCommand_ARM := UINT_TO_WORD(AI_Pusk_TH_faza_command);

  algoritms.Prov_PMS_ALG.inCommand_ARM := UINT_TO_WORD(AI_Prov_PMS_ALG_command);

  algoritms.Prov_opressovka_ALG.inCommand_ARM := UINT_TO_WORD(AI_Prov_opressovka_ALG_command);

  algoritms.Pusk_SEC_faza_chastotny.inCommand_ARM := UINT_TO_WORD(AI_Pusk_SEC_faza_chastotny_command);

  algoritms.Pusk_SEC_faza_reactor.inCommand_ARM := UINT_TO_WORD(AI_Pusk_SEC_faza_reactor_command);
END_FUNCTION_BLOCK

FUNCTION_BLOCK OPC_AI_SET
  VAR_EXTERNAL
    AI_Tstali_statora_kanal_1_HL : LREAL;
    AI_Tstali_statora_kanal_1_LL : LREAL;
    AI_Tstali_statora_kanal_1_command : UINT;
    AI_Tstali_statora_kanal_1_newHL : LREAL;
    AI_Tstali_statora_kanal_1_newLL : LREAL;
    AI_Tstali_statora_kanal_1_status : UDINT;
    AI_Tstali_statora_kanal_1_value : LREAL;
    AI_Tstali_statora_kanal_1_HW : LREAL;
    AI_Tstali_statora_kanal_1_newHW : LREAL;
    AI_Tstali_statora_kanal_2_HL : LREAL;
    AI_Tstali_statora_kanal_2_LL : LREAL;
    AI_Tstali_statora_kanal_2_command : UINT;
    AI_Tstali_statora_kanal_2_newHL : LREAL;
    AI_Tstali_statora_kanal_2_newLL : LREAL;
    AI_Tstali_statora_kanal_2_status : UDINT;
    AI_Tstali_statora_kanal_2_value : LREAL;
    AI_Tstali_statora_kanal_2_HW : LREAL;
    AI_Tstali_statora_kanal_2_newHW : LREAL;
    AI_Tstali_statora_kanal_3_HL : LREAL;
    AI_Tstali_statora_kanal_3_LL : LREAL;
    AI_Tstali_statora_kanal_3_command : UINT;
    AI_Tstali_statora_kanal_3_newHL : LREAL;
    AI_Tstali_statora_kanal_3_newLL : LREAL;
    AI_Tstali_statora_kanal_3_status : UDINT;
    AI_Tstali_statora_kanal_3_value : LREAL;
    AI_Tstali_statora_kanal_3_HW : LREAL;
    AI_Tstali_statora_kanal_3_newHW : LREAL;
    AI_Tmedi_statora_kanal_1_HL : LREAL;
    AI_Tmedi_statora_kanal_1_LL : LREAL;
    AI_Tmedi_statora_kanal_1_command : UINT;
    AI_Tmedi_statora_kanal_1_newHL : LREAL;
    AI_Tmedi_statora_kanal_1_newLL : LREAL;
    AI_Tmedi_statora_kanal_1_status : UDINT;
    AI_Tmedi_statora_kanal_1_value : LREAL;
    AI_Tmedi_statora_kanal_1_HW : LREAL;
    AI_Tmedi_statora_kanal_1_newHW : LREAL;
    AI_Tmedi_statora_kanal_2_HL : LREAL;
    AI_Tmedi_statora_kanal_2_LL : LREAL;
    AI_Tmedi_statora_kanal_2_command : UINT;
    AI_Tmedi_statora_kanal_2_newHL : LREAL;
    AI_Tmedi_statora_kanal_2_newLL : LREAL;
    AI_Tmedi_statora_kanal_2_status : UDINT;
    AI_Tmedi_statora_kanal_2_value : LREAL;
    AI_Tmedi_statora_kanal_2_HW : LREAL;
    AI_Tmedi_statora_kanal_2_newHW : LREAL;
    AI_Tmedi_statora_kanal_3_HL : LREAL;
    AI_Tmedi_statora_kanal_3_LL : LREAL;
    AI_Tmedi_statora_kanal_3_command : UINT;
    AI_Tmedi_statora_kanal_3_newHL : LREAL;
    AI_Tmedi_statora_kanal_3_newLL : LREAL;
    AI_Tmedi_statora_kanal_3_status : UDINT;
    AI_Tmedi_statora_kanal_3_value : LREAL;
    AI_Tmedi_statora_kanal_3_HW : LREAL;
    AI_Tmedi_statora_kanal_3_newHW : LREAL;
    AI_Toporno_podshipnika_EDT_1_HL : LREAL;
    AI_Toporno_podshipnika_EDT_1_LL : LREAL;
    AI_Toporno_podshipnika_EDT_1_command : UINT;
    AI_Toporno_podshipnika_EDT_1_newHL : LREAL;
    AI_Toporno_podshipnika_EDT_1_newLL : LREAL;
    AI_Toporno_podshipnika_EDT_1_status : UDINT;
    AI_Toporno_podshipnika_EDT_1_value : LREAL;
    AI_Toporno_podshipnika_EDT_1_HW : LREAL;
    AI_Toporno_podshipnika_EDT_1_newHW : LREAL;
    AI_Toporno_podshipnika_EDT_1_HA : LREAL;
    AI_Toporno_podshipnika_EDT_1_newHA : LREAL;
    AI_Toy_podshipnika_EDT_2_HL : LREAL;
    AI_Toy_podshipnika_EDT_2_LL : LREAL;
    AI_Toy_podshipnika_EDT_2_command : UINT;
    AI_Toy_podshipnika_EDT_2_newHL : LREAL;
    AI_Toy_podshipnika_EDT_2_newLL : LREAL;
    AI_Toy_podshipnika_EDT_2_status : UDINT;
    AI_Toy_podshipnika_EDT_2_value : LREAL;
    AI_Toy_podshipnika_EDT_2_HW : LREAL;
    AI_Toy_podshipnika_EDT_2_newHW : LREAL;
    AI_Toy_podshipnika_EDT_2_HA : LREAL;
    AI_Toy_podshipnika_EDT_2_newHA : LREAL;
    AI_Toy_podshipnika_kol_EDT_3_HL : LREAL;
    AI_Toy_podshipnika_kol_EDT_3_LL : LREAL;
    AI_Toy_podshipnika_kol_EDT_3_command : UINT;
    AI_Toy_podshipnika_kol_EDT_3_newHL : LREAL;
    AI_Toy_podshipnika_kol_EDT_3_newLL : LREAL;
    AI_Toy_podshipnika_kol_EDT_3_status : UDINT;
    AI_Toy_podshipnika_kol_EDT_3_value : LREAL;
    AI_Toy_podshipnika_kol_EDT_3_HW : LREAL;
    AI_Toy_podshipnika_kol_EDT_3_newHW : LREAL;
    AI_Toy_podshipnika_kol_EDT_3_HA : LREAL;
    AI_Toy_podshipnika_kol_EDT_3_newHA : LREAL;
    AI_Toy_podshipnika_kol_EDT_4_HL : LREAL;
    AI_Toy_podshipnika_kol_EDT_4_LL : LREAL;
    AI_Toy_podshipnika_kol_EDT_4_command : UINT;
    AI_Toy_podshipnika_kol_EDT_4_newHL : LREAL;
    AI_Toy_podshipnika_kol_EDT_4_newLL : LREAL;
    AI_Toy_podshipnika_kol_EDT_4_status : UDINT;
    AI_Toy_podshipnika_kol_EDT_4_value : LREAL;
    AI_Toy_podshipnika_kol_EDT_4_HW : LREAL;
    AI_Toy_podshipnika_kol_EDT_4_newHW : LREAL;
    AI_Toy_podshipnika_kol_EDT_4_HA : LREAL;
    AI_Toy_podshipnika_kol_EDT_4_newHA : LREAL;
    AI_Toy_podshipnika_shest_red_EDT_5_HL : LREAL;
    AI_Toy_podshipnika_shest_red_EDT_5_LL : LREAL;
    AI_Toy_podshipnika_shest_red_EDT_5_command : UINT;
    AI_Toy_podshipnika_shest_red_EDT_5_newHL : LREAL;
    AI_Toy_podshipnika_shest_red_EDT_5_newLL : LREAL;
    AI_Toy_podshipnika_shest_red_EDT_5_status : UDINT;
    AI_Toy_podshipnika_shest_red_EDT_5_value : LREAL;
    AI_Toy_podshipnika_shest_red_EDT_5_HW : LREAL;
    AI_Toy_podshipnika_shest_red_EDT_5_newHW : LREAL;
    AI_Toy_podshipnika_shest_red_EDT_5_HA : LREAL;
    AI_Toy_podshipnika_shest_red_EDT_5_newHA : LREAL;
    AI_Ty_podshipnika_red_EDT_6_HL : LREAL;
    AI_Ty_podshipnika_red_EDT_6_LL : LREAL;
    AI_Ty_podshipnika_red_EDT_6_command : UINT;
    AI_Ty_podshipnika_red_EDT_6_newHL : LREAL;
    AI_Ty_podshipnika_red_EDT_6_newLL : LREAL;
    AI_Ty_podshipnika_red_EDT_6_status : UDINT;
    AI_Ty_podshipnika_red_EDT_6_value : LREAL;
    AI_Ty_podshipnika_red_EDT_6_HW : LREAL;
    AI_Ty_podshipnika_red_EDT_6_newHW : LREAL;
    AI_Ty_podshipnika_red_EDT_6_HA : LREAL;
    AI_Ty_podshipnika_red_EDT_6_newHA : LREAL;
    AI_Ty_podshipnika_nagnet_EDT_7_1_HL : LREAL;
    AI_Ty_podshipnika_nagnet_EDT_7_1_LL : LREAL;
    AI_Ty_podshipnika_nagnet_EDT_7_1_command : UINT;
    AI_Ty_podshipnika_nagnet_EDT_7_1_newHL : LREAL;
    AI_Ty_podshipnika_nagnet_EDT_7_1_newLL : LREAL;
    AI_Ty_podshipnika_nagnet_EDT_7_1_status : UDINT;
    AI_Ty_podshipnika_nagnet_EDT_7_1_value : LREAL;
    AI_Ty_podshipnika_nagnet_EDT_7_1_HW : LREAL;
    AI_Ty_podshipnika_nagnet_EDT_7_1_newHW : LREAL;
    AI_Ty_podshipnika_nagnet_EDT_7_1_HA : LREAL;
    AI_Ty_podshipnika_nagnet_EDT_7_1_newHA : LREAL;
    AI_Ty_podshipnika_nagnet_EDT_7_2_HL : LREAL;
    AI_Ty_podshipnika_nagnet_EDT_7_2_LL : LREAL;
    AI_Ty_podshipnika_nagnet_EDT_7_2_command : UINT;
    AI_Ty_podshipnika_nagnet_EDT_7_2_newHL : LREAL;
    AI_Ty_podshipnika_nagnet_EDT_7_2_newLL : LREAL;
    AI_Ty_podshipnika_nagnet_EDT_7_2_status : UDINT;
    AI_Ty_podshipnika_nagnet_EDT_7_2_value : LREAL;
    AI_Ty_podshipnika_nagnet_EDT_7_2_HW : LREAL;
    AI_Ty_podshipnika_nagnet_EDT_7_2_newHW : LREAL;
    AI_Ty_podshipnika_nagnet_EDT_7_2_HA : LREAL;
    AI_Ty_podshipnika_nagnet_EDT_7_2_newHA : LREAL;
    AI_Toy_podshipnika_svobod_konca_EDT_8_1_HL : LREAL;
    AI_Toy_podshipnika_svobod_konca_EDT_8_1_LL : LREAL;
    AI_Toy_podshipnika_svobod_konca_EDT_8_1_command : UINT;
    AI_Toy_podshipnika_svobod_konca_EDT_8_1_newHL : LREAL;
    AI_Toy_podshipnika_svobod_konca_EDT_8_1_newLL : LREAL;
    AI_Toy_podshipnika_svobod_konca_EDT_8_1_status : UDINT;
    AI_Toy_podshipnika_svobod_konca_EDT_8_1_value : LREAL;
    AI_Toy_podshipnika_svobod_konca_EDT_8_1_HW : LREAL;
    AI_Toy_podshipnika_svobod_konca_EDT_8_1_newHW : LREAL;
    AI_Toy_podshipnika_svobod_konca_EDT_8_1_HA : LREAL;
    AI_Toy_podshipnika_svobod_konca_EDT_8_1_newHA : LREAL;
    AI_Toy_podshipnika_svobod_konca_EDT_8_2_HL : LREAL;
    AI_Toy_podshipnika_svobod_konca_EDT_8_2_LL : LREAL;
    AI_Toy_podshipnika_svobod_konca_EDT_8_2_command : UINT;
    AI_Toy_podshipnika_svobod_konca_EDT_8_2_newHL : LREAL;
    AI_Toy_podshipnika_svobod_konca_EDT_8_2_newLL : LREAL;
    AI_Toy_podshipnika_svobod_konca_EDT_8_2_status : UDINT;
    AI_Toy_podshipnika_svobod_konca_EDT_8_2_value : LREAL;
    AI_Toy_podshipnika_svobod_konca_EDT_8_2_HW : LREAL;
    AI_Toy_podshipnika_svobod_konca_EDT_8_2_newHW : LREAL;
    AI_Toy_podshipnika_svobod_konca_EDT_8_2_HA : LREAL;
    AI_Toy_podshipnika_svobod_konca_EDT_8_2_newHA : LREAL;
    AI_Toy_podshipnika_rab_kol_EDT_9_1_HL : LREAL;
    AI_Toy_podshipnika_rab_kol_EDT_9_1_LL : LREAL;
    AI_Toy_podshipnika_rab_kol_EDT_9_1_command : UINT;
    AI_Toy_podshipnika_rab_kol_EDT_9_1_newHL : LREAL;
    AI_Toy_podshipnika_rab_kol_EDT_9_1_newLL : LREAL;
    AI_Toy_podshipnika_rab_kol_EDT_9_1_status : UDINT;
    AI_Toy_podshipnika_rab_kol_EDT_9_1_value : LREAL;
    AI_Toy_podshipnika_rab_kol_EDT_9_1_HW : LREAL;
    AI_Toy_podshipnika_rab_kol_EDT_9_1_newHW : LREAL;
    AI_Toy_podshipnika_rab_kol_EDT_9_1_HA : LREAL;
    AI_Toy_podshipnika_rab_kol_EDT_9_1_newHA : LREAL;
    AI_Toy_podshipnika_rab_kol_EDT_9_2_HL : LREAL;
    AI_Toy_podshipnika_rab_kol_EDT_9_2_LL : LREAL;
    AI_Toy_podshipnika_rab_kol_EDT_9_2_command : UINT;
    AI_Toy_podshipnika_rab_kol_EDT_9_2_newHL : LREAL;
    AI_Toy_podshipnika_rab_kol_EDT_9_2_newLL : LREAL;
    AI_Toy_podshipnika_rab_kol_EDT_9_2_status : UDINT;
    AI_Toy_podshipnika_rab_kol_EDT_9_2_value : LREAL;
    AI_Toy_podshipnika_rab_kol_EDT_9_2_HW : LREAL;
    AI_Toy_podshipnika_rab_kol_EDT_9_2_newHW : LREAL;
    AI_Toy_podshipnika_rab_kol_EDT_9_2_HA : LREAL;
    AI_Toy_podshipnika_rab_kol_EDT_9_2_newHA : LREAL;
    AI_Toy_podshipnika_nerab_kol_EDT_10_1_HL : LREAL;
    AI_Toy_podshipnika_nerab_kol_EDT_10_1_LL : LREAL;
    AI_Toy_podshipnika_nerab_kol_EDT_10_1_command : UINT;
    AI_Toy_podshipnika_nerab_kol_EDT_10_1_newHL : LREAL;
    AI_Toy_podshipnika_nerab_kol_EDT_10_1_newLL : LREAL;
    AI_Toy_podshipnika_nerab_kol_EDT_10_1_status : UDINT;
    AI_Toy_podshipnika_nerab_kol_EDT_10_1_value : LREAL;
    AI_Toy_podshipnika_nerab_kol_EDT_10_1_HW : LREAL;
    AI_Toy_podshipnika_nerab_kol_EDT_10_1_newHW : LREAL;
    AI_Toy_podshipnika_nerab_kol_EDT_10_1_HA : LREAL;
    AI_Toy_podshipnika_nerab_kol_EDT_10_1_newHA : LREAL;
    AI_Toy_podshipnika_nerab_kol_EDT_10_2_HL : LREAL;
    AI_Toy_podshipnika_nerab_kol_EDT_10_2_LL : LREAL;
    AI_Toy_podshipnika_nerab_kol_EDT_10_2_command : UINT;
    AI_Toy_podshipnika_nerab_kol_EDT_10_2_newHL : LREAL;
    AI_Toy_podshipnika_nerab_kol_EDT_10_2_newLL : LREAL;
    AI_Toy_podshipnika_nerab_kol_EDT_10_2_status : UDINT;
    AI_Toy_podshipnika_nerab_kol_EDT_10_2_value : LREAL;
    AI_Toy_podshipnika_nerab_kol_EDT_10_2_HW : LREAL;
    AI_Toy_podshipnika_nerab_kol_EDT_10_2_newHW : LREAL;
    AI_Toy_podshipnika_nerab_kol_EDT_10_2_HA : LREAL;
    AI_Toy_podshipnika_nerab_kol_EDT_10_2_newHA : LREAL;
    AI_Tholodnogo_vozduha_ED_kanal_1_HL : LREAL;
    AI_Tholodnogo_vozduha_ED_kanal_1_LL : LREAL;
    AI_Tholodnogo_vozduha_ED_kanal_1_command : UINT;
    AI_Tholodnogo_vozduha_ED_kanal_1_newHL : LREAL;
    AI_Tholodnogo_vozduha_ED_kanal_1_newLL : LREAL;
    AI_Tholodnogo_vozduha_ED_kanal_1_status : UDINT;
    AI_Tholodnogo_vozduha_ED_kanal_1_value : LREAL;
    AI_Tholodnogo_vozduha_ED_kanal_1_HW : LREAL;
    AI_Tholodnogo_vozduha_ED_kanal_1_newHW : LREAL;
    AI_Tholodnogo_vozduha_ED_kanal_2_HL : LREAL;
    AI_Tholodnogo_vozduha_ED_kanal_2_LL : LREAL;
    AI_Tholodnogo_vozduha_ED_kanal_2_command : UINT;
    AI_Tholodnogo_vozduha_ED_kanal_2_newHL : LREAL;
    AI_Tholodnogo_vozduha_ED_kanal_2_newLL : LREAL;
    AI_Tholodnogo_vozduha_ED_kanal_2_status : UDINT;
    AI_Tholodnogo_vozduha_ED_kanal_2_value : LREAL;
    AI_Tholodnogo_vozduha_ED_kanal_2_HW : LREAL;
    AI_Tholodnogo_vozduha_ED_kanal_2_newHW : LREAL;
    AI_Tgorjachego_vozduha_ED_kanal_1_HL : LREAL;
    AI_Tgorjachego_vozduha_ED_kanal_1_LL : LREAL;
    AI_Tgorjachego_vozduha_ED_kanal_1_command : UINT;
    AI_Tgorjachego_vozduha_ED_kanal_1_newHL : LREAL;
    AI_Tgorjachego_vozduha_ED_kanal_1_newLL : LREAL;
    AI_Tgorjachego_vozduha_ED_kanal_1_status : UDINT;
    AI_Tgorjachego_vozduha_ED_kanal_1_value : LREAL;
    AI_Tgorjachego_vozduha_ED_kanal_1_HW : LREAL;
    AI_Tgorjachego_vozduha_ED_kanal_1_newHW : LREAL;
    AI_Tgorjachego_vozduha_ED_kanal_2_HL : LREAL;
    AI_Tgorjachego_vozduha_ED_kanal_2_LL : LREAL;
    AI_Tgorjachego_vozduha_ED_kanal_2_command : UINT;
    AI_Tgorjachego_vozduha_ED_kanal_2_newHL : LREAL;
    AI_Tgorjachego_vozduha_ED_kanal_2_newLL : LREAL;
    AI_Tgorjachego_vozduha_ED_kanal_2_status : UDINT;
    AI_Tgorjachego_vozduha_ED_kanal_2_value : LREAL;
    AI_Tgorjachego_vozduha_ED_kanal_2_HW : LREAL;
    AI_Tgorjachego_vozduha_ED_kanal_2_newHW : LREAL;
    AI_Tnarujnogo_vozduha_HL : LREAL;
    AI_Tnarujnogo_vozduha_LL : LREAL;
    AI_Tnarujnogo_vozduha_command : UINT;
    AI_Tnarujnogo_vozduha_newHL : LREAL;
    AI_Tnarujnogo_vozduha_newLL : LREAL;
    AI_Tnarujnogo_vozduha_status : UDINT;
    AI_Tnarujnogo_vozduha_value : LREAL;
    AI_Tnarujnogo_vozduha_HW : LREAL;
    AI_Tnarujnogo_vozduha_newHW : LREAL;
    AI_Tgaza_na_vhode_H_HL : LREAL;
    AI_Tgaza_na_vhode_H_LL : LREAL;
    AI_Tgaza_na_vhode_H_command : UINT;
    AI_Tgaza_na_vhode_H_newHL : LREAL;
    AI_Tgaza_na_vhode_H_newLL : LREAL;
    AI_Tgaza_na_vhode_H_status : UDINT;
    AI_Tgaza_na_vhode_H_value : LREAL;
    AI_Tgaza_na_vhode_H_HW : LREAL;
    AI_Tgaza_na_vhode_H_newHW : LREAL;
    AI_Tgaza_na_vyhode_H_HL : LREAL;
    AI_Tgaza_na_vyhode_H_LL : LREAL;
    AI_Tgaza_na_vyhode_H_command : UINT;
    AI_Tgaza_na_vyhode_H_newHL : LREAL;
    AI_Tgaza_na_vyhode_H_newLL : LREAL;
    AI_Tgaza_na_vyhode_H_status : UDINT;
    AI_Tgaza_na_vyhode_H_value : LREAL;
    AI_Tgaza_na_vyhode_H_HW : LREAL;
    AI_Tgaza_na_vyhode_H_newHW : LREAL;
    AI_Tgaza_na_vyhode_H_HA : LREAL;
    AI_Tgaza_na_vyhode_H_newHA : LREAL;
    AI_Tmasla_do_AVOM_HL : LREAL;
    AI_Tmasla_do_AVOM_LL : LREAL;
    AI_Tmasla_do_AVOM_command : UINT;
    AI_Tmasla_do_AVOM_newHL : LREAL;
    AI_Tmasla_do_AVOM_newLL : LREAL;
    AI_Tmasla_do_AVOM_status : UDINT;
    AI_Tmasla_do_AVOM_value : LREAL;
    AI_Tmasla_do_AVOM_HW : LREAL;
    AI_Tmasla_do_AVOM_newHW : LREAL;
    AI_Tmasla_posle_AVOM_HL : LREAL;
    AI_Tmasla_posle_AVOM_LL : LREAL;
    AI_Tmasla_posle_AVOM_command : UINT;
    AI_Tmasla_posle_AVOM_newHL : LREAL;
    AI_Tmasla_posle_AVOM_newLL : LREAL;
    AI_Tmasla_posle_AVOM_status : UDINT;
    AI_Tmasla_posle_AVOM_value : LREAL;
    AI_Tmasla_posle_AVOM_HW : LREAL;
    AI_Tmasla_posle_AVOM_newHW : LREAL;
    AI_Tmasla_MB_HL : LREAL;
    AI_Tmasla_MB_LL : LREAL;
    AI_Tmasla_MB_command : UINT;
    AI_Tmasla_MB_newHL : LREAL;
    AI_Tmasla_MB_newLL : LREAL;
    AI_Tmasla_MB_status : UDINT;
    AI_Tmasla_MB_value : LREAL;
    AI_Tmasla_MB_LW : LREAL;
    AI_Tmasla_MB_newLW : LREAL;
    AI_Tmasla_MB_TEN_HL : LREAL;
    AI_Tmasla_MB_TEN_LL : LREAL;
    AI_Tmasla_MB_TEN_command : UINT;
    AI_Tmasla_MB_TEN_newHL : LREAL;
    AI_Tmasla_MB_TEN_newLL : LREAL;
    AI_Tmasla_MB_TEN_status : UDINT;
    AI_Tmasla_MB_TEN_value : LREAL;
    AI_Tmasla_MB_TEN_HW : LREAL;
    AI_Tmasla_MB_TEN_newHW : LREAL;
    AI_Tshu_HL : LREAL;
    AI_Tshu_LL : LREAL;
    AI_Tshu_command : UINT;
    AI_Tshu_newHL : LREAL;
    AI_Tshu_newLL : LREAL;
    AI_Tshu_status : UDINT;
    AI_Tshu_value : LREAL;
    AI_Pmaslo_sm_nizkoe_HL : LREAL;
    AI_Pmaslo_sm_nizkoe_LL : LREAL;
    AI_Pmaslo_sm_nizkoe_command : UINT;
    AI_Pmaslo_sm_nizkoe_newHL : LREAL;
    AI_Pmaslo_sm_nizkoe_newLL : LREAL;
    AI_Pmaslo_sm_nizkoe_status : UDINT;
    AI_Pmaslo_sm_nizkoe_value : LREAL;
    AI_Pmaslo_sm_nizkoe_LW : LREAL;
    AI_Pmaslo_sm_nizkoe_newLW : LREAL;
    AI_Pmaslo_sm_nizkoe_LA : LREAL;
    AI_Pmaslo_sm_nizkoe_newLA : LREAL;
    AI_Pmaslo_sm_vysokoe_HL : LREAL;
    AI_Pmaslo_sm_vysokoe_LL : LREAL;
    AI_Pmaslo_sm_vysokoe_command : UINT;
    AI_Pmaslo_sm_vysokoe_newHL : LREAL;
    AI_Pmaslo_sm_vysokoe_newLL : LREAL;
    AI_Pmaslo_sm_vysokoe_status : UDINT;
    AI_Pmaslo_sm_vysokoe_value : LREAL;
    AI_Pmaslo_sm_vysokoe_LW : LREAL;
    AI_Pmaslo_sm_vysokoe_newLW : LREAL;
    AI_Pmaslo_sm_vysokoe_LA : LREAL;
    AI_Pmaslo_sm_vysokoe_newLA : LREAL;
    AI_Pmasla_posle_GNS_HL : LREAL;
    AI_Pmasla_posle_GNS_LL : LREAL;
    AI_Pmasla_posle_GNS_command : UINT;
    AI_Pmasla_posle_GNS_newHL : LREAL;
    AI_Pmasla_posle_GNS_newLL : LREAL;
    AI_Pmasla_posle_GNS_status : UDINT;
    AI_Pmasla_posle_GNS_value : LREAL;
    AI_Pmasla_posle_GNS_HW : LREAL;
    AI_Pmasla_posle_GNS_newHW : LREAL;
    AI_Pmasla_posle_GNS_LW : LREAL;
    AI_Pmasla_posle_GNS_newLW : LREAL;
    AI_Pmasla_posle_NU_HL : LREAL;
    AI_Pmasla_posle_NU_LL : LREAL;
    AI_Pmasla_posle_NU_command : UINT;
    AI_Pmasla_posle_NU_newHL : LREAL;
    AI_Pmasla_posle_NU_newLL : LREAL;
    AI_Pmasla_posle_NU_status : UDINT;
    AI_Pmasla_posle_NU_value : LREAL;
    AI_Pmasla_posle_NU_LW : LREAL;
    AI_Pmasla_posle_NU_newLW : LREAL;
    AI_Pgaza_na_vhode_nagnetatelia_HL : LREAL;
    AI_Pgaza_na_vhode_nagnetatelia_LL : LREAL;
    AI_Pgaza_na_vhode_nagnetatelia_command : UINT;
    AI_Pgaza_na_vhode_nagnetatelia_newHL : LREAL;
    AI_Pgaza_na_vhode_nagnetatelia_newLL : LREAL;
    AI_Pgaza_na_vhode_nagnetatelia_status : UDINT;
    AI_Pgaza_na_vhode_nagnetatelia_value : LREAL;
    AI_Pgaza_na_vhode_nagnetatelia_LW : LREAL;
    AI_Pgaza_na_vhode_nagnetatelia_newLW : LREAL;
    AI_Pgaza_na_vyhode_nagnetatelia_HL : LREAL;
    AI_Pgaza_na_vyhode_nagnetatelia_LL : LREAL;
    AI_Pgaza_na_vyhode_nagnetatelia_command : UINT;
    AI_Pgaza_na_vyhode_nagnetatelia_newHL : LREAL;
    AI_Pgaza_na_vyhode_nagnetatelia_newLL : LREAL;
    AI_Pgaza_na_vyhode_nagnetatelia_status : UDINT;
    AI_Pgaza_na_vyhode_nagnetatelia_value : LREAL;
    AI_Pgaza_na_vyhode_nagnetatelia_HW : LREAL;
    AI_Pgaza_na_vyhode_nagnetatelia_newHW : LREAL;
    AI_Pgaza_na_vyhode_nagnetatelia_HA : LREAL;
    AI_Pgaza_na_vyhode_nagnetatelia_newHA : LREAL;
    AI_Pimpuls_gaz_HL : LREAL;
    AI_Pimpuls_gaz_LL : LREAL;
    AI_Pimpuls_gaz_command : UINT;
    AI_Pimpuls_gaz_newHL : LREAL;
    AI_Pimpuls_gaz_newLL : LREAL;
    AI_Pimpuls_gaz_status : UDINT;
    AI_Pimpuls_gaz_value : LREAL;
    AI_Pimpuls_gaz_LW : LREAL;
    AI_Pimpuls_gaz_newLW : LREAL;
    AI_dPgaza_na_maslo_filtre_HL : LREAL;
    AI_dPgaza_na_maslo_filtre_LL : LREAL;
    AI_dPgaza_na_maslo_filtre_command : UINT;
    AI_dPgaza_na_maslo_filtre_newHL : LREAL;
    AI_dPgaza_na_maslo_filtre_newLL : LREAL;
    AI_dPgaza_na_maslo_filtre_status : UDINT;
    AI_dPgaza_na_maslo_filtre_value : LREAL;
    AI_dPgaza_na_maslo_filtre_HW : LREAL;
    AI_dPgaza_na_maslo_filtre_newHW : LREAL;
    AI_dPgaza_na_konfuzore_HL : LREAL;
    AI_dPgaza_na_konfuzore_LL : LREAL;
    AI_dPgaza_na_konfuzore_command : UINT;
    AI_dPgaza_na_konfuzore_newHL : LREAL;
    AI_dPgaza_na_konfuzore_newLL : LREAL;
    AI_dPgaza_na_konfuzore_status : UDINT;
    AI_dPgaza_na_konfuzore_value : LREAL;
    AI_dPgaza_na_konfuzore_LW : LREAL;
    AI_dPgaza_na_konfuzore_newLW : LREAL;
    AI_dPmaslo_gaz_HL : LREAL;
    AI_dPmaslo_gaz_LL : LREAL;
    AI_dPmaslo_gaz_command : UINT;
    AI_dPmaslo_gaz_newHL : LREAL;
    AI_dPmaslo_gaz_newLL : LREAL;
    AI_dPmaslo_gaz_status : UDINT;
    AI_dPmaslo_gaz_value : LREAL;
    AI_dPmaslo_gaz_LW : LREAL;
    AI_dPmaslo_gaz_newLW : LREAL;
    AI_dPmaslo_gaz_LA : LREAL;
    AI_dPmaslo_gaz_newLA : LREAL;
    AI_Os_sdvig_nagnetatelja_plus_HL : LREAL;
    AI_Os_sdvig_nagnetatelja_plus_LL : LREAL;
    AI_Os_sdvig_nagnetatelja_plus_command : UINT;
    AI_Os_sdvig_nagnetatelja_plus_newHL : LREAL;
    AI_Os_sdvig_nagnetatelja_plus_newLL : LREAL;
    AI_Os_sdvig_nagnetatelja_plus_status : UDINT;
    AI_Os_sdvig_nagnetatelja_plus_value : LREAL;
    AI_Os_sdvig_nagnetatelja_plus_HW : LREAL;
    AI_Os_sdvig_nagnetatelja_plus_newHW : LREAL;
    AI_Os_sdvig_nagnetatelja_plus_HA : LREAL;
    AI_Os_sdvig_nagnetatelja_plus_newHA : LREAL;
    AI_Os_sdvig_nagnetatelja_minus_HL : LREAL;
    AI_Os_sdvig_nagnetatelja_minus_LL : LREAL;
    AI_Os_sdvig_nagnetatelja_minus_command : UINT;
    AI_Os_sdvig_nagnetatelja_minus_newHL : LREAL;
    AI_Os_sdvig_nagnetatelja_minus_newLL : LREAL;
    AI_Os_sdvig_nagnetatelja_minus_status : UDINT;
    AI_Os_sdvig_nagnetatelja_minus_value : LREAL;
    AI_Os_sdvig_nagnetatelja_minus_LW : LREAL;
    AI_Os_sdvig_nagnetatelja_minus_newLW : LREAL;
    AI_Os_sdvig_nagnetatelja_minus_LA : LREAL;
    AI_Os_sdvig_nagnetatelja_minus_newLA : LREAL;
    AI_Yroven_masla_MB_HL : LREAL;
    AI_Yroven_masla_MB_LL : LREAL;
    AI_Yroven_masla_MB_command : UINT;
    AI_Yroven_masla_MB_newHL : LREAL;
    AI_Yroven_masla_MB_newLL : LREAL;
    AI_Yroven_masla_MB_status : UDINT;
    AI_Yroven_masla_MB_value : LREAL;
    AI_Yroven_masla_MB_LW : LREAL;
    AI_Yroven_masla_MB_newLW : LREAL;
    AI_Kontrol_per_220V_HL : LREAL;
    AI_Kontrol_per_220V_LL : LREAL;
    AI_Kontrol_per_220V_command : UINT;
    AI_Kontrol_per_220V_newHL : LREAL;
    AI_Kontrol_per_220V_newLL : LREAL;
    AI_Kontrol_per_220V_status : UDINT;
    AI_Kontrol_per_220V_value : LREAL;
    AI_Kontrol_per_220V_HW : LREAL;
    AI_Kontrol_per_220V_newHW : LREAL;
    AI_Kontrol_per_220V_LW : LREAL;
    AI_Kontrol_per_220V_newLW : LREAL;
    AI_Kontrol_post_220V_HL : LREAL;
    AI_Kontrol_post_220V_LL : LREAL;
    AI_Kontrol_post_220V_command : UINT;
    AI_Kontrol_post_220V_newHL : LREAL;
    AI_Kontrol_post_220V_newLL : LREAL;
    AI_Kontrol_post_220V_status : UDINT;
    AI_Kontrol_post_220V_value : LREAL;
    AI_Kontrol_post_220V_HW : LREAL;
    AI_Kontrol_post_220V_newHW : LREAL;
    AI_Kontrol_post_220V_LW : LREAL;
    AI_Kontrol_post_220V_newLW : LREAL;
    AI_Tok_statora_HL : LREAL;
    AI_Tok_statora_LL : LREAL;
    AI_Tok_statora_command : UINT;
    AI_Tok_statora_newHL : LREAL;
    AI_Tok_statora_newLL : LREAL;
    AI_Tok_statora_status : UDINT;
    AI_Tok_statora_value : LREAL;
    AI_Tok_statora_LW : LREAL;
    AI_Tok_statora_newLW : LREAL;
    AI_Vibro_skorost_OPED_T1_HL : LREAL;
    AI_Vibro_skorost_OPED_T1_LL : LREAL;
    AI_Vibro_skorost_OPED_T1_command : UINT;
    AI_Vibro_skorost_OPED_T1_newHL : LREAL;
    AI_Vibro_skorost_OPED_T1_newLL : LREAL;
    AI_Vibro_skorost_OPED_T1_status : UDINT;
    AI_Vibro_skorost_OPED_T1_value : LREAL;
    AI_Vibro_skorost_OPED_T1_HW : LREAL;
    AI_Vibro_skorost_OPED_T1_newHW : LREAL;
    AI_Vibro_skorost_OPED_T1_HA : LREAL;
    AI_Vibro_skorost_OPED_T1_newHA : LREAL;
    AI_Vibro_skorost_OYPED_T2_HL : LREAL;
    AI_Vibro_skorost_OYPED_T2_LL : LREAL;
    AI_Vibro_skorost_OYPED_T2_command : UINT;
    AI_Vibro_skorost_OYPED_T2_newHL : LREAL;
    AI_Vibro_skorost_OYPED_T2_newLL : LREAL;
    AI_Vibro_skorost_OYPED_T2_status : UDINT;
    AI_Vibro_skorost_OYPED_T2_value : LREAL;
    AI_Vibro_skorost_OYPED_T2_HW : LREAL;
    AI_Vibro_skorost_OYPED_T2_newHW : LREAL;
    AI_Vibro_skorost_OYPED_T2_HA : LREAL;
    AI_Vibro_skorost_OYPED_T2_newHA : LREAL;
    AI_Vibro_skorost_OYP_kolesa_ED_T3_HL : LREAL;
    AI_Vibro_skorost_OYP_kolesa_ED_T3_LL : LREAL;
    AI_Vibro_skorost_OYP_kolesa_ED_T3_command : UINT;
    AI_Vibro_skorost_OYP_kolesa_ED_T3_newHL : LREAL;
    AI_Vibro_skorost_OYP_kolesa_ED_T3_newLL : LREAL;
    AI_Vibro_skorost_OYP_kolesa_ED_T3_status : UDINT;
    AI_Vibro_skorost_OYP_kolesa_ED_T3_value : LREAL;
    AI_Vibro_skorost_OYP_kolesa_ED_T3_HW : LREAL;
    AI_Vibro_skorost_OYP_kolesa_ED_T3_newHW : LREAL;
    AI_Vibro_skorost_OYP_kolesa_ED_T3_HA : LREAL;
    AI_Vibro_skorost_OYP_kolesa_ED_T3_newHA : LREAL;
    AI_Vibro_skorost_OP_kolesa_RH_T4_HL : LREAL;
    AI_Vibro_skorost_OP_kolesa_RH_T4_LL : LREAL;
    AI_Vibro_skorost_OP_kolesa_RH_T4_command : UINT;
    AI_Vibro_skorost_OP_kolesa_RH_T4_newHL : LREAL;
    AI_Vibro_skorost_OP_kolesa_RH_T4_newLL : LREAL;
    AI_Vibro_skorost_OP_kolesa_RH_T4_status : UDINT;
    AI_Vibro_skorost_OP_kolesa_RH_T4_value : LREAL;
    AI_Vibro_skorost_OP_kolesa_RH_T4_HW : LREAL;
    AI_Vibro_skorost_OP_kolesa_RH_T4_newHW : LREAL;
    AI_Vibro_skorost_OP_kolesa_RH_T4_HA : LREAL;
    AI_Vibro_skorost_OP_kolesa_RH_T4_newHA : LREAL;
    AI_Vibro_skorost_OP_shesterni_RED_T5_HL : LREAL;
    AI_Vibro_skorost_OP_shesterni_RED_T5_LL : LREAL;
    AI_Vibro_skorost_OP_shesterni_RED_T5_command : UINT;
    AI_Vibro_skorost_OP_shesterni_RED_T5_newHL : LREAL;
    AI_Vibro_skorost_OP_shesterni_RED_T5_newLL : LREAL;
    AI_Vibro_skorost_OP_shesterni_RED_T5_status : UDINT;
    AI_Vibro_skorost_OP_shesterni_RED_T5_value : LREAL;
    AI_Vibro_skorost_OP_shesterni_RED_T5_HW : LREAL;
    AI_Vibro_skorost_OP_shesterni_RED_T5_newHW : LREAL;
    AI_Vibro_skorost_OP_shesterni_RED_T5_HA : LREAL;
    AI_Vibro_skorost_OP_shesterni_RED_T5_newHA : LREAL;
    AI_Vibro_skorost_OP_shesterni_RED_T6_HL : LREAL;
    AI_Vibro_skorost_OP_shesterni_RED_T6_LL : LREAL;
    AI_Vibro_skorost_OP_shesterni_RED_T6_command : UINT;
    AI_Vibro_skorost_OP_shesterni_RED_T6_newHL : LREAL;
    AI_Vibro_skorost_OP_shesterni_RED_T6_newLL : LREAL;
    AI_Vibro_skorost_OP_shesterni_RED_T6_status : UDINT;
    AI_Vibro_skorost_OP_shesterni_RED_T6_value : LREAL;
    AI_Vibro_skorost_OP_shesterni_RED_T6_HW : LREAL;
    AI_Vibro_skorost_OP_shesterni_RED_T6_newHW : LREAL;
    AI_Vibro_skorost_OP_shesterni_RED_T6_HA : LREAL;
    AI_Vibro_skorost_OP_shesterni_RED_T6_newHA : LREAL;
  END_VAR
